// TwinCAT 3 PLC project MistralPLC
// ProgramVersion: 3.1.4023.0
// libraries:
//   Tc2_FTP, * (Beckhoff Automation GmbH)
//   Tc2_Standard, * (Beckhoff Automation GmbH)
//   Tc2_System, * (Beckhoff Automation GmbH)
//   Tc2_TcpIp, * (Beckhoff Automation GmbH)
//   Tc2_Utilities, * (Beckhoff Automation GmbH)
//   Tc3_EventLogger, * (Beckhoff Automation GmbH)
//   Tc3_Module, * (Beckhoff Automation GmbH)
//   Util, * (System)
// project tree:
//   Data types/ E_ClientSteps.TcDUT, E_DataExchaSteps.TcDUT
//   DUTs/ ST_LoadData.TcDUT
//   GVLs/Conveyor_1/ GVL_bButt_1.TcGVL, GVL_bDriveReady_1.TcGVL, GVL_bDrive_1.TcGVL, GVL_bLongMove_1.TcGVL, GVL_bMove_1.TcGVL, GVL_bPerm_1.TcGVL, GVL_bSens_1.TcGVL, GVL_BusyFree_1.TcGVL
//   GVLs/Conveyor_2/ GVL_bButt_2.TcGVL, GVL_bDriveReady_2.TcGVL, GVL_bDriveSpeed_2.TcGVL, GVL_bDrive_2.TcGVL, GVL_bLongMove_2.TcGVL, GVL_bMove_2.TcGVL, GVL_bPerm_2.TcGVL, GVL_bSens_2.TcGVL, GVL_BusyFree_2.TcGVL
//   GVLs/Conveyor_3/ GVL_bButt_3.TcGVL, GVL_bDriveReady_3.TcGVL, GVL_bDriveSpeed_3.TcGVL, GVL_bDrive_3.TcGVL, GVL_bLongMove_3.TcGVL, GVL_bMove_3.TcGVL, GVL_bPerm_3.TcGVL, GVL_bSens_3.TcGVL, GVL_BusyFree_3.TcGVL
//   GVLs/Conveyor_4/ GVL_bButt_4.TcGVL, GVL_bDriveReady_4.TcGVL, GVL_bDriveSpeed_4.TcGVL, GVL_bDrive_4.TcGVL, GVL_bLongMove_4.TcGVL, GVL_bMove_4.TcGVL, GVL_bPerm_4.TcGVL, GVL_bSens_4.TcGVL, GVL_BusyFree_4.TcGVL
//   GVLs/ Global_Variables.TcGVL, GVL.TcGVL, GVL_Alarm.TcGVL, GVL_Lights.TcGVL, GVL_LoadData_1.TcGVL
//   / PlcTask.TcTTO
//   POUs/Alarms/ AlarmEventGeneral.TcPOU, AlarmEvent_conv1.TcPOU, AlarmEvent_conv2.TcPOU, AlarmEvent_conv3.TcPOU, AlarmEvent_conv4.TcPOU, Alarm_conv_1.TcPOU, Alarm_conv_2.TcPOU, Alarm_conv_3.TcPOU, Alarm_conv_4.TcPOU, Alarm_conv_General.TcPOU, FB_AlarmEvent.TcPOU
//   POUs/ ConvLine1.TcPOU, ConvLine2.TcPOU, ConvLine3.TcPOU, ConvLine4.TcPOU, MAIN.TcPOU, TCP_IP.TcPOU
//   POUs/Ethernet/ FB_Server.TcPOU, FB_ServerApplication.TcPOU, FB_ServerConnection.TcPOU
//   POUs/Ethernet/Helper POUs/ FB_FrameFifo.TcPOU, FB_LogFifo.TcPOU
//   POUs/ExchangeWMS/ Exchange_WMS.TcPOU, FB_CreateMessage.TcPOU, FB_LoadDataToWMS.TcPOU, FB_Tail.TcPOU, FB_TransBuffer.TcPOU, FB_Upload_ToServer.TcPOU
//   POUs/FB/FBauxiliary/ FB_Busy1.TcPOU, FB_Busy2.TcPOU, FB_ButtonToggle.TcPOU
//   POUs/FB/FBconv/ FB_ConvPlace.TcPOU, FB_ConvPlaceDouble.TcPOU
//   POUs/FB/ FB_Direction.TcPOU, FB_Puls.TcPOU, Puls.TcPOU
//   POUs/ProcessingLoadData/ FB_LoadScan.TcPOU, FB_LoadWeight.TcPOU
// real-time tasks:
//   TASK PlcTask: cycle T#10ms, priority 20, ADS port 350
// I/O:
//   DEVICE Device 2 (Profinet Controller CCAT (RT)), AmsNetId 5.79.109.88.2.1
//     scale1 [BIZERBA BIZERBA Industrial weighing terminal WM4 920008000]
//       modules: Term 1 (DAP Module), Term 2 (Output 1 word), Term 3 (Output 1 byte), Term 4 (Output 1 byte), Term 5 (Output 1 byte), Term 6 (Output 1 byte), Term 7 (Output 1 byte), Term 8 (Output 1 byte), Term 9 (Output 1 byte), Term 10 (Output 1 byte), Term 11 (Output 1 byte), Term 12 (Output 1 byte), Term 13 (Output 1 byte), Term 14 (Output 1 byte), Term 15 (Output 1 byte), Term 16 (Output 1 byte), Term 17 (Input 1 word), Term 18 (Input 2 word), Term 19 (Input 1 byte), Term 20 (Input 1 byte), Term 21 (Input 1 byte), Term 22 (Input 1 byte), Term 23 (Input 1 byte), Term 24 (Input 1 byte), Term 25 (Input 1 byte), Term 26 (Input 1 byte), Term 27 (Input 1 byte), Term 28 (Input 1 byte)
//     scale2 [BIZERBA BIZERBA Industrial weighing terminal WM4 920008000]
//       modules: Term 31 (DAP Module), Term 86 (Output 1 word), Term 87 (Output 1 byte), Term 88 (Output 1 byte), Term 89 (Output 1 byte), Term 90 (Output 1 byte), Term 91 (Output 1 byte), Term 92 (Output 1 byte), Term 93 (Output 1 byte), Term 94 (Output 1 byte), Term 95 (Output 1 byte), Term 96 (Output 1 byte), Term 97 (Output 1 byte), Term 98 (Output 1 byte), Term 99 (Output 1 byte), Term 100 (Output 1 byte), Term 101 (Input 1 word), Term 102 (Input 2 word), Term 103 (Input 1 byte), Term 104 (Input 1 byte), Term 105 (Input 1 byte), Term 106 (Input 1 byte), Term 107 (Input 1 byte), Term 108 (Input 1 byte), Term 109 (Input 1 byte), Term 110 (Input 1 byte), Term 111 (Input 1 byte), Term 112 (Input 1 byte)
//     scale3 [BIZERBA BIZERBA Industrial weighing terminal WM4 920008000]
//       modules: Term 29 (DAP Module), Term 32 (Output 1 word), Term 33 (Output 1 byte), Term 34 (Output 1 byte), Term 35 (Output 1 byte), Term 36 (Output 1 byte), Term 37 (Output 1 byte), Term 38 (Output 1 byte), Term 39 (Output 1 byte), Term 40 (Output 1 byte), Term 41 (Output 1 byte), Term 42 (Output 1 byte), Term 43 (Output 1 byte), Term 44 (Output 1 byte), Term 45 (Output 1 byte), Term 46 (Output 1 byte), Term 47 (Input 1 word), Term 48 (Input 2 word), Term 49 (Input 1 byte), Term 50 (Input 1 byte), Term 51 (Input 1 byte), Term 52 (Input 1 byte), Term 53 (Input 1 byte), Term 54 (Input 1 byte), Term 55 (Input 1 byte), Term 56 (Input 1 byte), Term 57 (Input 1 byte), Term 58 (Input 1 byte)
//     scale4 [BIZERBA BIZERBA Industrial weighing terminal WM4 920008000]
//       modules: Term 30 (DAP Module), Term 59 (Output 1 word), Term 60 (Output 1 byte), Term 61 (Output 1 byte), Term 62 (Output 1 byte), Term 63 (Output 1 byte), Term 64 (Output 1 byte), Term 65 (Output 1 byte), Term 66 (Output 1 byte), Term 67 (Output 1 byte), Term 68 (Output 1 byte), Term 69 (Output 1 byte), Term 70 (Output 1 byte), Term 71 (Output 1 byte), Term 72 (Output 1 byte), Term 73 (Output 1 byte), Term 74 (Input 1 word), Term 75 (Input 2 word), Term 76 (Input 1 byte), Term 77 (Input 1 byte), Term 78 (Input 1 byte), Term 79 (Input 1 byte), Term 80 (Input 1 byte), Term 81 (Input 1 byte), Term 82 (Input 1 byte), Term 83 (Input 1 byte), Term 84 (Input 1 byte), Term 85 (Input 1 byte)
//   DEVICE Device 1 (EtherCAT), AmsNetId 5.79.109.88.3.1
//     Term 1 (EK1200) [EK1200-5000 EtherCAT Power supply (2A E-Bus)]
//       Term 2 (EL1008) [EL1008 8Ch. Dig. Input 24V, 3ms]
//       Term 3 (EL1008) [EL1008 8Ch. Dig. Input 24V, 3ms]
//       Term 4 (EL1008) [EL1008 8Ch. Dig. Input 24V, 3ms]
//       Term 5 (EL1008) [EL1008 8Ch. Dig. Input 24V, 3ms]
//       Term 6 (EL1008) [EL1008 8Ch. Dig. Input 24V, 3ms]
//       Term 7 (EL2008) [EL2008 8Ch. Dig. Output 24V, 0.5A]
//       Term 8 (EL2008) [EL2008 8Ch. Dig. Output 24V, 0.5A]
//       Term 9 (EL2008) [EL2008 8Ch. Dig. Output 24V, 0.5A]
//       Term 10 (EL2008) [EL2008 8Ch. Dig. Output 24V, 0.5A]
//       Term 11 (EK1122) [EK1122 2 port EtherCAT junction]
//         Term 12 (EK1100) [EK1100 EtherCAT Coupler (2A E-Bus)]
//           Term 15 (EL1008) [EL1008 8Ch. Dig. Input 24V, 3ms]
//           Term 16 (EL1008) [EL1008 8Ch. Dig. Input 24V, 3ms]
//           Term 17 (EL1008) [EL1008 8Ch. Dig. Input 24V, 3ms]
//           Term 18 (EL1008) [EL1008 8Ch. Dig. Input 24V, 3ms]
//           Term 19 (EL1008) [EL1008 8Ch. Dig. Input 24V, 3ms]
//           Term 20 (EL2008) [EL2008 8Ch. Dig. Output 24V, 0.5A]
//           Term 21 (EL2008) [EL2008 8Ch. Dig. Output 24V, 0.5A]
//           Term 22 (EL2008) [EL2008 8Ch. Dig. Output 24V, 0.5A]
//           Term 23 (EL2008) [EL2008 8Ch. Dig. Output 24V, 0.5A]
//           Term 24 (EK1322) [EK1322 2-port EtherCAT P junction with feed-in]
//             Box 1 (EPP2339-0021) X3 [EPP2339-0021 16 Ch. Dig. Input/Output 24V, 0,5A, M8]
//             Box 2 (EPP1004-0061) X3 [EPP1004-0061 4 Ch. Dig. Input 24V, 3ms, M8]
//             Box 3 (EPP2339-0021) X3 [EPP2339-0021 16 Ch. Dig. Input/Output 24V, 0,5A, M8]
//             Box 4 (EPP2339-0021) X4 [EPP2339-0021 16 Ch. Dig. Input/Output 24V, 0,5A, M8]
//             Box 5 (EPP1004-0061) X4 [EPP1004-0061 4 Ch. Dig. Input 24V, 3ms, M8]
//             Box 6 (EPP2339-0021) X4 [EPP2339-0021 16 Ch. Dig. Input/Output 24V, 0,5A, M8]
//       Term 13 (EK1322) [EK1322 2-port EtherCAT P junction with feed-in]
//         Box 1 (EPP2339-0021) X1 [EPP2339-0021 16 Ch. Dig. Input/Output 24V, 0,5A, M8]
//         Box 2 (EPP1004-0061) X1 [EPP1004-0061 4 Ch. Dig. Input 24V, 3ms, M8]
//         Box 3 (EPP2339-0021) X1 [EPP2339-0021 16 Ch. Dig. Input/Output 24V, 0,5A, M8]
//         Box 4 (EPP2339-0021) X2 [EPP2339-0021 16 Ch. Dig. Input/Output 24V, 0,5A, M8]
//         Box 5 (EPP1004-0061) X2 [EPP1004-0061 4 Ch. Dig. Input 24V, 3ms, M8]
//         Box 6 (EPP2339-0021) X2 [EPP2339-0021 16 Ch. Dig. Input/Output 24V, 0,5A, M8]
// variable links:
//   MistralPLC/MistralPLC Instance <-> Device 1 (EtherCAT)/Term 1 (EK1200)/Term 11 (EK1122)/Term 12 (EK1100)/Term 15 (EL1008)
//     PlcTask Inputs/GVL.b_3AS1 <-> Channel 3/Input
//     PlcTask Inputs/GVL.b_4AS1 <-> Channel 4/Input
//     PlcTask Inputs/GVL.b_K2_ <-> Channel 2/Input
//     PlcTask Inputs/GVL.b_SF3_ <-> Channel 1/Input
//   MistralPLC/MistralPLC Instance <-> Device 1 (EtherCAT)/Term 1 (EK1200)/Term 11 (EK1122)/Term 12 (EK1100)/Term 16 (EL1008)
//     PlcTask Inputs/GVL.b_3KM1_1 <-> Channel 2/Input
//     PlcTask Inputs/GVL.b_3KM1_2 <-> Channel 3/Input
//     PlcTask Inputs/GVL.b_4KM1_1 <-> Channel 5/Input
//     PlcTask Inputs/GVL.b_4KM1_2 <-> Channel 6/Input
//     PlcTask Inputs/GVL.b_3QF1 <-> Channel 1/Input
//     PlcTask Inputs/GVL.b_4QF1 <-> Channel 4/Input
//   MistralPLC/MistralPLC Instance <-> Device 1 (EtherCAT)/Term 1 (EK1200)/Term 11 (EK1122)/Term 12 (EK1100)/Term 17 (EL1008)
//     PlcTask Inputs/GVL.b_3KM{2..7} <-> Channel {3..8}/Input  (6 links)
//     PlcTask Inputs/GVL.b_3QF2_3QF7 <-> Channel 1/Input
//     PlcTask Inputs/GVL.b_3QF8 <-> Channel 2/Input
//   MistralPLC/MistralPLC Instance <-> Device 1 (EtherCAT)/Term 1 (EK1200)/Term 11 (EK1122)/Term 12 (EK1100)/Term 18 (EL1008)
//     PlcTask Inputs/GVL.b_4KM{2..7} <-> Channel {3..8}/Input  (6 links)
//     PlcTask Inputs/GVL.b_4QF2_4QF7 <-> Channel 1/Input
//     PlcTask Inputs/GVL.b_4QF8 <-> Channel 2/Input
//   MistralPLC/MistralPLC Instance <-> Device 1 (EtherCAT)/Term 1 (EK1200)/Term 11 (EK1122)/Term 12 (EK1100)/Term 20 (EL2008)
//     PlcTask Outputs/GVL.b3K{2..5} <-> Channel {5..8}/Output  (4 links)
//     PlcTask Outputs/GVL.b_3K1_1 <-> Channel 1/Output
//     PlcTask Outputs/GVL.b_3K1_2 <-> Channel 2/Output
//     PlcTask Outputs/GVL.b_4K1_1 <-> Channel 3/Output
//     PlcTask Outputs/GVL.b_4K1_2 <-> Channel 4/Output
//   MistralPLC/MistralPLC Instance <-> Device 1 (EtherCAT)/Term 1 (EK1200)/Term 11 (EK1122)/Term 12 (EK1100)/Term 21 (EL2008)
//     PlcTask Outputs/GVL.b3K6 <-> Channel 1/Output
//     PlcTask Outputs/GVL.b3K7 <-> Channel 2/Output
//     PlcTask Outputs/GVL.b4K2 <-> Channel 3/Output
//     PlcTask Outputs/GVL.b4K3 <-> Channel 4/Output
//     PlcTask Outputs/GVL.b4K4 <-> Channel 5/Output
//     PlcTask Outputs/GVL.b4K5 <-> Channel 6/Output
//     PlcTask Outputs/GVL.b4K6 <-> Channel 7/Output
//     PlcTask Outputs/GVL.b4K7 <-> Channel 8/Output
//   MistralPLC/MistralPLC Instance <-> Device 1 (EtherCAT)/Term 1 (EK1200)/Term 11 (EK1122)/Term 12 (EK1100)/Term 22 (EL2008)
//     PlcTask Outputs/GVL.b2Sh_SB0 <-> Channel 5/Output
//     PlcTask Outputs/GVL.b2Sh_SB1 <-> Channel 6/Output
//     PlcTask Outputs/GVL.b3S1_SB0 <-> Channel 1/Output
//     PlcTask Outputs/GVL.b3S6_SB0 <-> Channel 2/Output
//     PlcTask Outputs/GVL.b4S1_SB0 <-> Channel 3/Output
//     PlcTask Outputs/GVL.b4S6_SB0 <-> Channel 4/Output
//   MistralPLC/MistralPLC Instance <-> Device 1 (EtherCAT)/Term 1 (EK1200)/Term 11 (EK1122)/Term 12 (EK1100)/Term 24 (EK1322)/Box 1 (EPP2339-0021) X3
//     PlcTask Inputs/GVL.b3_S6_SB0 <-> Channel 11/Input
//     PlcTask Inputs/GVL_bSens_3.bSens3s04D1 <-> Channel 1/Input
//     PlcTask Inputs/GVL_bSens_3.bSens3s04D2 <-> Channel 2/Input
//     PlcTask Inputs/GVL_bSens_3.bSens3s04D3 <-> Channel 3/Input
//     PlcTask Inputs/GVL_bSens_3.bSens3s05D1 <-> Channel 4/Input
//     PlcTask Inputs/GVL_bSens_3.bSens3s05D2 <-> Channel 5/Input
//     PlcTask Inputs/GVL_bSens_3.bSens3s06D1 <-> Channel 6/Input
//     PlcTask Inputs/GVL_bSens_3.bSens3s06D2 <-> Channel 7/Input
//     PlcTask Outputs/GVL.b_3S4_2A2 <-> Channel 25/Output
//     PlcTask Outputs/GVL.b_3S5_2A1 <-> Channel 26/Output
//     PlcTask Outputs/GVL_Lights.bBlue_3S1HL1 <-> Channel 32/Output
//     PlcTask Outputs/GVL_Lights.bGreen_3S1HL1 <-> Channel 30/Output
//     PlcTask Outputs/GVL_Lights.bRed_3S1HL1 <-> Channel 29/Output
//     PlcTask Outputs/GVL_Lights.bSound_3S1HL1 <-> Channel 28/Output
//     PlcTask Outputs/GVL_Lights.bYellow_3S1HL1 <-> Channel 31/Output
//   MistralPLC/MistralPLC Instance <-> Device 1 (EtherCAT)/Term 1 (EK1200)/Term 11 (EK1122)/Term 12 (EK1100)/Term 24 (EK1322)/Box 2 (EPP1004-0061) X3
//     PlcTask Inputs/GVL_bSens_3.bSens3s02D1 <-> Channel 1/Input
//     PlcTask Inputs/GVL_bSens_3.bSens3s02D2 <-> Channel 2/Input
//     PlcTask Inputs/GVL_bSens_3.bSens3s03D1 <-> Channel 3/Input
//     PlcTask Inputs/GVL_bSens_3.bSens3s03D2 <-> Channel 4/Input
//   MistralPLC/MistralPLC Instance <-> Device 1 (EtherCAT)/Term 1 (EK1200)/Term 11 (EK1122)/Term 12 (EK1100)/Term 24 (EK1322)/Box 3 (EPP2339-0021) X3
//     PlcTask Inputs/GVL.b3_S1_SB0 <-> Channel 9/Input
//     PlcTask Inputs/GVL_bSens_3.bSens3s01D1 <-> Channel 1/Input
//     PlcTask Inputs/GVL_bSens_3.bSens3s01D2 <-> Channel 2/Input
//     PlcTask Inputs/GVL_bSens_3.bSens3s01D3 <-> Channel 3/Input
//     PlcTask Outputs/GVL_Lights.bBlue_3S1_HL1 <-> Channel 24/Output
//     PlcTask Outputs/GVL_Lights.bGreen_3S1_HL1 <-> Channel 22/Output
//     PlcTask Outputs/GVL_Lights.bRed_3S1_HL1 <-> Channel 21/Output
//     PlcTask Outputs/GVL_Lights.bSound_3S1_HL1 <-> Channel 20/Output
//     PlcTask Outputs/GVL_Lights.bYellow_3S1_HL1 <-> Channel 23/Output
//   MistralPLC/MistralPLC Instance <-> Device 1 (EtherCAT)/Term 1 (EK1200)/Term 11 (EK1122)/Term 12 (EK1100)/Term 24 (EK1322)/Box 4 (EPP2339-0021) X4
//     PlcTask Inputs/GVL.b4_S6_SB0 <-> Channel 11/Input
//     PlcTask Inputs/GVL_bSens_4.bSens4s04D1 <-> Channel 1/Input
//     PlcTask Inputs/GVL_bSens_4.bSens4s04D2 <-> Channel 2/Input
//     PlcTask Inputs/GVL_bSens_4.bSens4s04D3 <-> Channel 3/Input
//     PlcTask Inputs/GVL_bSens_4.bSens4s05D1 <-> Channel 4/Input
//     PlcTask Inputs/GVL_bSens_4.bSens4s05D2 <-> Channel 5/Input
//     PlcTask Inputs/GVL_bSens_4.bSens4s06D1 <-> Channel 6/Input
//     PlcTask Inputs/GVL_bSens_4.bSens4s06D2 <-> Channel 7/Input
//     PlcTask Outputs/GVL.b_4S4_2A2 <-> Channel 25/Output
//     PlcTask Outputs/GVL.b_4S5_2A1 <-> Channel 26/Output
//     PlcTask Outputs/GVL_Lights.bBlue_4S1HL1 <-> Channel 32/Output
//     PlcTask Outputs/GVL_Lights.bGreen_4S1HL1 <-> Channel 30/Output
//     PlcTask Outputs/GVL_Lights.bRed_4S1HL1 <-> Channel 24/Output
//     PlcTask Outputs/GVL_Lights.bSound_4S1HL1 <-> Channel 28/Output
//     PlcTask Outputs/GVL_Lights.bYellow_4S1HL1 <-> Channel 31/Output
//   MistralPLC/MistralPLC Instance <-> Device 1 (EtherCAT)/Term 1 (EK1200)/Term 11 (EK1122)/Term 12 (EK1100)/Term 24 (EK1322)/Box 5 (EPP1004-0061) X4
//     PlcTask Inputs/GVL_bSens_4.bSens4s02D1 <-> Channel 1/Input
//     PlcTask Inputs/GVL_bSens_4.bSens4s02D2 <-> Channel 2/Input
//     PlcTask Inputs/GVL_bSens_4.bSens4s03D1 <-> Channel 3/Input
//     PlcTask Inputs/GVL_bSens_4.bSens4s03D2 <-> Channel 4/Input
//   MistralPLC/MistralPLC Instance <-> Device 1 (EtherCAT)/Term 1 (EK1200)/Term 11 (EK1122)/Term 12 (EK1100)/Term 24 (EK1322)/Box 6 (EPP2339-0021) X4
//     PlcTask Inputs/GVL.b4_S1_SB0 <-> Channel 9/Input
//     PlcTask Inputs/GVL_bSens_4.bSens4s01D1 <-> Channel 1/Input
//     PlcTask Inputs/GVL_bSens_4.bSens4s01D2 <-> Channel 2/Input
//     PlcTask Inputs/GVL_bSens_4.bSens4s01D3 <-> Channel 3/Input
//     PlcTask Outputs/GVL_Lights.bBlue_4S1_HL1 <-> Channel 24/Output
//     PlcTask Outputs/GVL_Lights.bGreen_4S1_HL1 <-> Channel 22/Output
//     PlcTask Outputs/GVL_Lights.bRed_4S1_HL1 <-> Channel 21/Output
//     PlcTask Outputs/GVL_Lights.bSound_4S1_HL1 <-> Channel 20/Output
//     PlcTask Outputs/GVL_Lights.bYellow_4S1_HL1 <-> Channel 23/Output
//   MistralPLC/MistralPLC Instance <-> Device 1 (EtherCAT)/Term 1 (EK1200)/Term 13 (EK1322)/Box 1 (EPP2339-0021) X1
//     PlcTask Inputs/GVL.b1_S6_SB0 <-> Channel 11/Input
//     PlcTask Inputs/GVL_bSens_1.bSens1s04D1 <-> Channel 1/Input
//     PlcTask Inputs/GVL_bSens_1.bSens1s04D2 <-> Channel 2/Input
//     PlcTask Inputs/GVL_bSens_1.bSens1s04D3 <-> Channel 3/Input
//     PlcTask Inputs/GVL_bSens_1.bSens1s05D1 <-> Channel 4/Input
//     PlcTask Inputs/GVL_bSens_1.bSens1s05D2 <-> Channel 5/Input
//     PlcTask Inputs/GVL_bSens_1.bSens1s06D1 <-> Channel 6/Input
//     PlcTask Inputs/GVL_bSens_1.bSens1s06D2 <-> Channel 7/Input
//     PlcTask Outputs/GVL.b_1S4_2A2 <-> Channel 25/Output
//     PlcTask Outputs/GVL.b_1S5_2A1 <-> Channel 26/Output
//     PlcTask Outputs/GVL_Lights.bBlue_1S1HL1 <-> Channel 32/Output
//     PlcTask Outputs/GVL_Lights.bGreen_1S1HL1 <-> Channel 30/Output
//     PlcTask Outputs/GVL_Lights.bRed_1S1HL1 <-> Channel 29/Output
//     PlcTask Outputs/GVL_Lights.bSound_1S1HL1 <-> Channel 28/Output
//     PlcTask Outputs/GVL_Lights.bYellow_1S1HL1 <-> Channel 31/Output
//   MistralPLC/MistralPLC Instance <-> Device 1 (EtherCAT)/Term 1 (EK1200)/Term 13 (EK1322)/Box 2 (EPP1004-0061) X1
//     PlcTask Inputs/GVL_bSens_1.bSens1s02D1 <-> Channel 1/Input
//     PlcTask Inputs/GVL_bSens_1.bSens1s02D2 <-> Channel 2/Input
//     PlcTask Inputs/GVL_bSens_1.bSens1s03D1 <-> Channel 3/Input
//     PlcTask Inputs/GVL_bSens_1.bSens1s03D2 <-> Channel 4/Input
//   MistralPLC/MistralPLC Instance <-> Device 1 (EtherCAT)/Term 1 (EK1200)/Term 13 (EK1322)/Box 3 (EPP2339-0021) X1
//     PlcTask Inputs/GVL.b1_S1_SB0 <-> Channel 9/Input
//     PlcTask Inputs/GVL_bSens_1.bSens1s01D1 <-> Channel 1/Input
//     PlcTask Inputs/GVL_bSens_1.bSens1s01D2 <-> Channel 2/Input
//     PlcTask Inputs/GVL_bSens_1.bSens1s01D3 <-> Channel 3/Input
//     PlcTask Outputs/GVL_Lights.bBlue_1S1_HL1 <-> Channel 24/Output
//     PlcTask Outputs/GVL_Lights.bGreen_1S1_HL1 <-> Channel 22/Output
//     PlcTask Outputs/GVL_Lights.bRed_1S1_HL1 <-> Channel 21/Output
//     PlcTask Outputs/GVL_Lights.bSound_1S1_HL1 <-> Channel 20/Output
//     PlcTask Outputs/GVL_Lights.bYellow_1S1_HL1 <-> Channel 23/Output
//   MistralPLC/MistralPLC Instance <-> Device 1 (EtherCAT)/Term 1 (EK1200)/Term 13 (EK1322)/Box 4 (EPP2339-0021) X2
//     PlcTask Inputs/GVL.b2_S6_SB0 <-> Channel 11/Input
//     PlcTask Inputs/GVL_bSens_2.bSens2s04D1 <-> Channel 1/Input
//     PlcTask Inputs/GVL_bSens_2.bSens2s04D2 <-> Channel 2/Input
//     PlcTask Inputs/GVL_bSens_2.bSens2s04D3 <-> Channel 3/Input
//     PlcTask Inputs/GVL_bSens_2.bSens2s05D1 <-> Channel 4/Input
//     PlcTask Inputs/GVL_bSens_2.bSens2s05D2 <-> Channel 5/Input
//     PlcTask Inputs/GVL_bSens_2.bSens2s06D1 <-> Channel 6/Input
//     PlcTask Inputs/GVL_bSens_2.bSens2s06D2 <-> Channel 7/Input
//     PlcTask Outputs/GVL.b_2S4_2A2 <-> Channel 25/Output
//     PlcTask Outputs/GVL.b_2S5_2A1 <-> Channel 26/Output
//     PlcTask Outputs/GVL_Lights.bBlue_2S1HL1 <-> Channel 32/Output
//     PlcTask Outputs/GVL_Lights.bGreen_2S1HL1 <-> Channel 30/Output
//     PlcTask Outputs/GVL_Lights.bRed_2S1HL1 <-> Channel 29/Output
//     PlcTask Outputs/GVL_Lights.bSound_2S1HL1 <-> Channel 28/Output
//     PlcTask Outputs/GVL_Lights.bYellow_2S1HL1 <-> Channel 31/Output
//   MistralPLC/MistralPLC Instance <-> Device 1 (EtherCAT)/Term 1 (EK1200)/Term 13 (EK1322)/Box 5 (EPP1004-0061) X2
//     PlcTask Inputs/GVL_bSens_2.bSens2s02D1 <-> Channel 1/Input
//     PlcTask Inputs/GVL_bSens_2.bSens2s02D2 <-> Channel 2/Input
//     PlcTask Inputs/GVL_bSens_2.bSens2s03D1 <-> Channel 3/Input
//     PlcTask Inputs/GVL_bSens_2.bSens2s03D2 <-> Channel 4/Input
//   MistralPLC/MistralPLC Instance <-> Device 1 (EtherCAT)/Term 1 (EK1200)/Term 13 (EK1322)/Box 6 (EPP2339-0021) X2
//     PlcTask Inputs/GVL.b2_S1_SB0 <-> Channel 9/Input
//     PlcTask Inputs/GVL_bSens_2.bSens2s01D1 <-> Channel 1/Input
//     PlcTask Inputs/GVL_bSens_2.bSens2s01D2 <-> Channel 2/Input
//     PlcTask Inputs/GVL_bSens_2.bSens2s01D3 <-> Channel 3/Input
//     PlcTask Outputs/GVL_Lights.bBlue_2S1_HL1 <-> Channel 24/Output
//     PlcTask Outputs/GVL_Lights.bGreen_2S1_HL1 <-> Channel 22/Output
//     PlcTask Outputs/GVL_Lights.bRed_2S1_HL1 <-> Channel 21/Output
//     PlcTask Outputs/GVL_Lights.bSound_2S1_HL1 <-> Channel 20/Output
//     PlcTask Outputs/GVL_Lights.bYellow_2S1_HL1 <-> Channel 23/Output
//   MistralPLC/MistralPLC Instance <-> Device 1 (EtherCAT)/Term 1 (EK1200)/Term 2 (EL1008)
//     PlcTask Inputs/GVL.b_1AS1 <-> Channel 5/Input
//     PlcTask Inputs/GVL.b_2AS1 <-> Channel 6/Input
//     PlcTask Inputs/GVL.b_1QF <-> Channel 1/Input
//     PlcTask Inputs/GVL.b_2QF <-> Channel 2/Input
//     PlcTask Inputs/GVL.b_GP3 <-> Channel 7/Input
//     PlcTask Inputs/GVL.b_K2 <-> Channel 4/Input
//     PlcTask Inputs/GVL.b_SF3 <-> Channel 3/Input
//   MistralPLC/MistralPLC Instance <-> Device 1 (EtherCAT)/Term 1 (EK1200)/Term 3 (EL1008)
//     PlcTask Inputs/GVL.b_1KM1_1 <-> Channel 2/Input
//     PlcTask Inputs/GVL.b_1KM1_2 <-> Channel 3/Input
//     PlcTask Inputs/GVL.b_2KM1_1 <-> Channel 5/Input
//     PlcTask Inputs/GVL.b_2KM1_2 <-> Channel 6/Input
//     PlcTask Inputs/GVL.b_1P_I <-> Channel 7/Input
//     PlcTask Inputs/GVL.b_1P_U <-> Channel 8/Input
//     PlcTask Inputs/GVL.b_1QF1 <-> Channel 1/Input
//     PlcTask Inputs/GVL.b_2QF1 <-> Channel 4/Input
//   MistralPLC/MistralPLC Instance <-> Device 1 (EtherCAT)/Term 1 (EK1200)/Term 4 (EL1008)
//     PlcTask Inputs/GVL.b_1KM{2..7} <-> Channel {3..8}/Input  (6 links)
//     PlcTask Inputs/GVL.b_1QF2_1QF7 <-> Channel 1/Input
//     PlcTask Inputs/GVL.b_1QF8 <-> Channel 2/Input
//   MistralPLC/MistralPLC Instance <-> Device 1 (EtherCAT)/Term 1 (EK1200)/Term 5 (EL1008)
//     PlcTask Inputs/GVL.b_2KM{2..7} <-> Channel {3..8}/Input  (6 links)
//     PlcTask Inputs/GVL.b_2QF2_2QF7 <-> Channel 1/Input
//     PlcTask Inputs/GVL.b_2QF8 <-> Channel 2/Input
//   MistralPLC/MistralPLC Instance <-> Device 1 (EtherCAT)/Term 1 (EK1200)/Term 7 (EL2008)
//     PlcTask Outputs/GVL.b1K{2..5} <-> Channel {5..8}/Output  (4 links)
//     PlcTask Outputs/GVL.b_1K1_1 <-> Channel 1/Output
//     PlcTask Outputs/GVL.b_1K1_2 <-> Channel 2/Output
//     PlcTask Outputs/GVL.b_2K1_1 <-> Channel 3/Output
//     PlcTask Outputs/GVL.b_2K1_2 <-> Channel 4/Output
//   MistralPLC/MistralPLC Instance <-> Device 1 (EtherCAT)/Term 1 (EK1200)/Term 8 (EL2008)
//     PlcTask Outputs/GVL.b1K6 <-> Channel 1/Output
//     PlcTask Outputs/GVL.b1K7 <-> Channel 2/Output
//     PlcTask Outputs/GVL.b2K2 <-> Channel 3/Output
//     PlcTask Outputs/GVL.b2K3 <-> Channel 4/Output
//     PlcTask Outputs/GVL.b2K4 <-> Channel 5/Output
//     PlcTask Outputs/GVL.b2K5 <-> Channel 6/Output
//     PlcTask Outputs/GVL.b2K6 <-> Channel 7/Output
//     PlcTask Outputs/GVL.b2K7 <-> Channel 8/Output
//   MistralPLC/MistralPLC Instance <-> Device 1 (EtherCAT)/Term 1 (EK1200)/Term 9 (EL2008)
//     PlcTask Outputs/GVL.b1S1_SB0 <-> Channel 1/Output
//     PlcTask Outputs/GVL.b1S6_SB0 <-> Channel 2/Output
//     PlcTask Outputs/GVL.b2S1_SB0 <-> Channel 3/Output
//     PlcTask Outputs/GVL.b2S6_SB0 <-> Channel 4/Output
//     PlcTask Outputs/GVL.b1Sh_SB0 <-> Channel 5/Output
//     PlcTask Outputs/GVL.b1Sh_SB1 <-> Channel 6/Output
//   MistralPLC/MistralPLC Instance <-> Device 2 (Profinet Controller CCAT (RT))/scale1
//     PlcTask Inputs/GVL.Massa_1 <-> API/Term 18 (Input 2 word)/Subterm 21 (Input 2 word)/Inputs/Input
//   MistralPLC/MistralPLC Instance <-> Device 2 (Profinet Controller CCAT (RT))/scale2
//     PlcTask Inputs/GVL.Massa_2 <-> API/Term 102 (Input 2 word)/Subterm 114 (Input 2 word)/Inputs/Input
//   MistralPLC/MistralPLC Instance <-> Device 2 (Profinet Controller CCAT (RT))/scale3
//     PlcTask Inputs/GVL.Massa_3 <-> API/Term 48 (Input 2 word)/Subterm 60 (Input 2 word)/Inputs/Input
//   MistralPLC/MistralPLC Instance <-> Device 2 (Profinet Controller CCAT (RT))/scale4
//     PlcTask Inputs/GVL.Massa_4 <-> API/Term 75 (Input 2 word)/Subterm 87 (Input 2 word)/Inputs/Input

CONFIGURATION MistralPLC
    RESOURCE PLC ON TwinCAT3
        TASK PlcTask(INTERVAL := T#10ms, PRIORITY := 20);
        PROGRAM MAIN WITH PlcTask : MAIN;
    END_RESOURCE
END_CONFIGURATION

// ---- Data types/E_ClientSteps.TcDUT
TYPE E_ClientSteps :
(
	CLIENT_STATE_IDLE,
	CLIENT_STATE_CONNECT_START,
	CLIENT_STATE_CONNECT_WAIT,
	CLIENT_STATE_DATAEXCHA_START,
	CLIENT_STATE_DATAEXCHA_WAIT,
	CLIENT_STATE_CLOSE_START,
	CLIENT_STATE_CLOSE_WAIT,
	CLIENT_STATE_ERROR
);
END_TYPE

// ---- Data types/E_DataExchaSteps.TcDUT
TYPE E_DataExchaSteps :
(
	DATAEXCHA_STATE_IDLE,
	DATAEXCHA_STATE_SEND_START,
	DATAEXCHA_STATE_SEND_WAIT,
	DATAEXCHA_STATE_RECEIVE_START,
	DATAEXCHA_STATE_RECEIVE_WAIT,
	DATAEXCHA_STATE_ERROR
);
END_TYPE

// ---- DUTs/ST_LoadData.TcDUT
TYPE ST_LoadData :
STRUCT
	sID: STRING;
	sWeight: STRING;
END_STRUCT
END_TYPE

// ---- GVLs/Conveyor_1/GVL_bButt_1.TcGVL
VAR_GLOBAL
	bButtAuto1		:BOOL;
	bButtManu1		:BOOL;
	bButtStop1 		:BOOL;
	bButtReverse1 	:BOOL;
//-------------------------//
	bButt1s01		:BOOL;
	bButt1s01Rev	:BOOL;
	bButt1s02		:BOOL;
	bButt1s02Rev	:BOOL;
	bButt1s03		:BOOL;
	bButt1s03Rev	:BOOL;
	bButt1s04		:BOOL;
	bButt1s04Rev	:BOOL;								
	bButt1s05		:BOOL;									
	bButt1s05Rev	:BOOL;									
	bButt1s06		:BOOL;									
	bButt1s06Rev	:BOOL;
//-------------------------//
	bButt1s01_s02	:BOOL;
	bButt1s02_s03	:BOOL;
	bButt1s03_s04	:BOOL;
	bButt1s04_s05	:BOOL;
	bButt1s05_s06	:BOOL;

END_VAR

// ---- GVLs/Conveyor_1/GVL_bDriveReady_1.TcGVL
VAR_GLOBAL
// Готовность двигателей

bDriveReady1s01M1	AT%I* :BOOL;	// Конороль готовности конвейер 1 секция 1

bDriveReady1s02M1	AT%I* :BOOL;	// Конороль готовности конвейер 1 секция 2

bDriveReady1s03M1	AT%I* :BOOL;	// Конороль готовности конвейер 1 секция 3

bDriveReady1s04M1	AT%I* :BOOL;	// Конороль готовности конвейер 1 секция 4

bDriveReady1s05M1	AT%I* :BOOL;	// Конороль готовности конвейер 1 секция 5

bDriveReady1s06M1	AT%I* :BOOL;	// Конороль готовности конвейер 1 секция 6
END_VAR

// ---- GVLs/Conveyor_1/GVL_bDrive_1.TcGVL
VAR_GLOBAL

	bDrive1s01M1		  	 :BOOL;	
	bDrive1s01M1Rev	  		 :BOOL;

	bDrive1s02M1		  	 :BOOL;	
	bDrive1s02M1Rev	  		 :BOOL;

	bDrive1s03M1		  	 :BOOL;	
	bDrive1s03M1Rev	  		 :BOOL;

	bDrive1s04M1		  	 :BOOL;	
	bDrive1s04M1Rev	  		 :BOOL;

	bDrive1s05M1		  	 :BOOL;	
	bDrive1s05M1Rev	  		 :BOOL;

	bDrive1s06M1		  	 :BOOL;	
	bDrive1s06M1Rev	  		 :BOOL;
END_VAR

// ---- GVLs/Conveyor_1/GVL_bLongMove_1.TcGVL
VAR_GLOBAL
// Долгие перемещения
// Прямое движение	
bLongMove1s01_s02_1		:BOOL;
bLongMove1s02_1_s02_2   :BOOL;
bLongMove1s02_2_s03_1   :BOOL;
bLongMove1s02_s03       :BOOL;
bLongMove1s03_1_s03_2   :BOOL;
bLongMove1s03_2_s04_1   :BOOL;
bLongMove1s03_s04       :BOOL;
bLongMove1s04_1_s04_2   :BOOL;
bLongMove1s04_2_s05     :BOOL;
bLongMove1s05_1s06		:BOOL;

bLongMove_1s01_s02_1	 :BOOL;
bLongMove_1s02_1_s02_2   :BOOL;
bLongMove_1s02_2_s03_1   :BOOL;
bLongMove_1s02_s03       :BOOL;
bLongMove_1s03_1_s03_2   :BOOL;
bLongMove_1s03_2_s04_1   :BOOL;
bLongMove_1s03_s04       :BOOL;
bLongMove_1s04_1_s04_2   :BOOL;
bLongMove_1s04_2_s05     :BOOL;
bLongMove_1s05_1s06		:BOOL;  







END_VAR

// ---- GVLs/Conveyor_1/GVL_bMove_1.TcGVL
VAR_GLOBAL
// Прямое движение
bMove1s01_s02_1		:BOOL;
bMove1s02_1_s02_2	:BOOL;

bMove1s02_2_s03_1	:BOOL;
bMove1s02_s03		:BOOL;
bMove1s03_1_s03_2	:BOOL;

bMove1s03_2_s04_1	:BOOL;
bMove1s03_s04		:BOOL;
bMove1s04_1_s04_2	:BOOL;

bMove1s04_2_s05		:BOOL;
bMove1s05_s06		:BOOL;

END_VAR

// ---- GVLs/Conveyor_1/GVL_bPerm_1.TcGVL
VAR_GLOBAL
// Разрешение на движение
// Прямое движение
bPerm1s01_1s02	:BOOL;
bPerm1s02_1s03	:BOOL;
bPerm1s03_1s04	:BOOL;
bPerm1s04_1s05	:BOOL;
bPerm1s05_1s06	:BOOL;
// Обратное движение
bPerm1s06_1s05	:BOOL;
bPerm1s05_1s04	:BOOL;
bPerm1s04_1s03	:BOOL;
bPerm1s03_1s02	:BOOL;
bPerm1s02_1s01	:BOOL;
END_VAR

// ---- GVLs/Conveyor_1/GVL_bSens_1.TcGVL
VAR_GLOBAL
// --------------------------------------Список датчиков--------------------------------------------//
//---------------------------------------Первый конвейер--------------------------------------------//
{attribute 'TcLinkTo' := 'TIID^Device 1 (EtherCAT)^Term 1 (EK1200)^Term 13 (EK1322)^Box 3 (EPP2339-0021) X1^Channel 1^Input'}
bSens1s01D1 AT%I* :BOOL;	// Датчик в конце секции (в прямом направлении)
{attribute 'TcLinkTo' := 'TIID^Device 1 (EtherCAT)^Term 1 (EK1200)^Term 13 (EK1322)^Box 3 (EPP2339-0021) X1^Channel 2^Input'}
bSens1s01D2 AT%I* :BOOL;	// Датчик в конце секции (в обратном направлении)
{attribute 'TcLinkTo' := 'TIID^Device 1 (EtherCAT)^Term 1 (EK1200)^Term 13 (EK1322)^Box 3 (EPP2339-0021) X1^Channel 3^Input'}
bSens1s01D3 AT%I* :BOOL;	// Датчик контроля вил 
{attribute 'TcLinkTo' := 'TIID^Device 1 (EtherCAT)^Term 1 (EK1200)^Term 13 (EK1322)^Box 2 (EPP1004-0061) X1^Channel 1^Input'}
bSens1s02D1 AT%I* :BOOL;	// Датчик в конце секции (в прямом направлении)
{attribute 'TcLinkTo' := 'TIID^Device 1 (EtherCAT)^Term 1 (EK1200)^Term 13 (EK1322)^Box 2 (EPP1004-0061) X1^Channel 2^Input'}
bSens1s02D2 AT%I* :BOOL;	// Датчик в середине секции 
{attribute 'TcLinkTo' := 'TIID^Device 1 (EtherCAT)^Term 1 (EK1200)^Term 13 (EK1322)^Box 2 (EPP1004-0061) X1^Channel 3^Input'}
bSens1s03D1 AT%I* :BOOL;	// Датчик в конце секции (в прямом направлении)
{attribute 'TcLinkTo' := 'TIID^Device 1 (EtherCAT)^Term 1 (EK1200)^Term 13 (EK1322)^Box 2 (EPP1004-0061) X1^Channel 4^Input'}
bSens1s03D2 AT%I* :BOOL;	// Датчик в середине секции 
{attribute 'TcLinkTo' := 'TIID^Device 1 (EtherCAT)^Term 1 (EK1200)^Term 13 (EK1322)^Box 1 (EPP2339-0021) X1^Channel 1^Input'}
bSens1s04D1 AT%I* :BOOL;	// Датчик в конце секции (в прямом направлении)
{attribute 'TcLinkTo' := 'TIID^Device 1 (EtherCAT)^Term 1 (EK1200)^Term 13 (EK1322)^Box 1 (EPP2339-0021) X1^Channel 2^Input'}
bSens1s04D2 AT%I* :BOOL;	// Датчик в середине секции 
{attribute 'TcLinkTo' := 'TIID^Device 1 (EtherCAT)^Term 1 (EK1200)^Term 13 (EK1322)^Box 1 (EPP2339-0021) X1^Channel 3^Input'}
bSens1s04D3 AT%I* :BOOL;	// Датчик сканирования RFID
{attribute 'TcLinkTo' := 'TIID^Device 1 (EtherCAT)^Term 1 (EK1200)^Term 13 (EK1322)^Box 1 (EPP2339-0021) X1^Channel 4^Input'}
bSens1s05D1 AT%I* :BOOL;	// Датчик в конце секции (в прямом направлении)
{attribute 'TcLinkTo' := 'TIID^Device 1 (EtherCAT)^Term 1 (EK1200)^Term 13 (EK1322)^Box 1 (EPP2339-0021) X1^Channel 5^Input'}
bSens1s05D2 AT%I* :BOOL;	// Датчик управления двойным движением
{attribute 'TcLinkTo' := 'TIID^Device 1 (EtherCAT)^Term 1 (EK1200)^Term 13 (EK1322)^Box 1 (EPP2339-0021) X1^Channel 6^Input'}
bSens1s06D1 AT%I* :BOOL;	// Датчик в конце секции (в прямом направлении)
{attribute 'TcLinkTo' := 'TIID^Device 1 (EtherCAT)^Term 1 (EK1200)^Term 13 (EK1322)^Box 1 (EPP2339-0021) X1^Channel 7^Input'}
bSens1s06D2 AT%I* :BOOL;	// Датчик контроля вил

END_VAR

// ---- GVLs/Conveyor_1/GVL_BusyFree_1.TcGVL
VAR_GLOBAL
(*Текущее состояние платформы (Занято/Свободно)*)
(*Первый этаж*)
	bPlatformBusy1s01	 	:BOOL;
	bPlatformFree1s01 		:BOOL;
	bPlatformBusy1s02 		:BOOL;
	bPlatformFree1s02 		:BOOL;
	bPlatformBusy1s03 		:BOOL;
	bPlatformFree1s03 		:BOOL;
	bPlatformBusy1s04 		:BOOL;
	bPlatformFree1s04 		:BOOL;
	bPlatformBusy1s05		:BOOL;
	bPlatformFree1s05 		:BOOL;
	bPlatformBusy1s06		:BOOL;
	bPlatformFree1s06 		:BOOL;
END_VAR

// ---- GVLs/Conveyor_2/GVL_bButt_2.TcGVL
VAR_GLOBAL
	bButtAuto2		:BOOL;
	bButtManu2		:BOOL;
	bButtStop2 		:BOOL;
	bButtReverse2 	:BOOL;
//-------------------------//
	bButt2s01		:BOOL;
	bButt2s01Rev	:BOOL;
	bButt2s02		:BOOL;
	bButt2s02Rev	:BOOL;
	bButt2s03		:BOOL;
	bButt2s03Rev	:BOOL;
	bButt2s04		:BOOL;
	bButt2s04Rev	:BOOL;								
	bButt2s05		:BOOL;									
	bButt2s05Rev	:BOOL;									
	bButt2s06		:BOOL;									
	bButt2s06Rev	:BOOL;
//-------------------------//
	bButt2s01_s02	:BOOL;
	bButt2s02_s03	:BOOL;
	bButt2s03_s04	:BOOL;
	bButt2s04_s05	:BOOL;
	bButt2s05_s06	:BOOL;
END_VAR

// ---- GVLs/Conveyor_2/GVL_bDriveReady_2.TcGVL
VAR_GLOBAL
// Готовность двигателей

bDriveReady2s01M1	AT%I* :BOOL;	// Конороль готовности MoviMot конвейер 2 секция 1

bDriveReady2s02M1	AT%I* :BOOL;	// Конороль готовности MoviMot конвейер 2 секция 2

bDriveReady2s03M1	AT%I* :BOOL;	// Конороль готовности MoviMot конвейер 2 секция 3

bDriveReady2s04M1	AT%I* :BOOL;	// Конороль готовности MoviSwitch конвейер 2 секция 4

bDriveReady2s05M1	AT%I* :BOOL;	// Конороль готовности MoviSwitch конвейер 2 секция 5

bDriveReady2s06M1	AT%I* :BOOL;	// Конороль готовности MoviSwitch конвейер 2 секция 6
END_VAR

// ---- GVLs/Conveyor_2/GVL_bDriveSpeed_2.TcGVL
VAR_GLOBAL
// Включение второй скорости для секций

bDrive2s01Speed2			AT%Q* :BOOL;

bDrive2s02Speed2			AT%Q* :BOOL;

bDrive2s03Speed2			AT%Q* :BOOL;

bDrive2s04Speed2			AT%Q* :BOOL;

bDrive2s05Speed2			AT%Q* :BOOL;

bDrive2s06Speed2			AT%Q* :BOOL;
END_VAR

// ---- GVLs/Conveyor_2/GVL_bDrive_2.TcGVL
VAR_GLOBAL

	bDrive2s01M1		  	AT%Q* :BOOL;	
	bDrive2s01M1Rev	  		AT%Q* :BOOL;

	bDrive2s02M1		  	AT%Q* :BOOL;	
	bDrive2s02M1Rev	  		AT%Q* :BOOL;

	bDrive2s03M1		  	AT%Q* :BOOL;	
	bDrive2s03M1Rev	  		AT%Q* :BOOL;

	bDrive2s04M1		  	AT%Q* :BOOL;	
	bDrive2s04M1Rev	  		AT%Q* :BOOL;

	bDrive2s05M1		  	AT%Q* :BOOL;	
	bDrive2s05M1Rev	  		AT%Q* :BOOL;

	bDrive2s06M1		  	AT%Q* :BOOL;	
	bDrive2s06M1Rev	 	  	AT%Q* :BOOL;
END_VAR

// ---- GVLs/Conveyor_2/GVL_bLongMove_2.TcGVL
VAR_GLOBAL
// Долгие перемещения
// Прямое движение	
bLongMove2s01_s02_1		:BOOL;
bLongMove2s02_1_s02_2   :BOOL;
bLongMove2s02_2_s03_1   :BOOL;
bLongMove2s02_s03       :BOOL;
bLongMove2s03_1_s03_2   :BOOL;
bLongMove2s03_2_s04_1   :BOOL;
bLongMove2s03_s04       :BOOL;
bLongMove2s04_1_s04_2   :BOOL;
bLongMove2s04_2_s05     :BOOL;
bLongMove2s05_1s06		:BOOL;

bLongMove_2s01_s02_1	 :BOOL;
bLongMove_2s02_1_s02_2   :BOOL;
bLongMove_2s02_2_s03_1   :BOOL;
bLongMove_2s02_s03       :BOOL;
bLongMove_2s03_1_s03_2   :BOOL;
bLongMove_2s03_2_s04_1   :BOOL;
bLongMove_2s03_s04       :BOOL;
bLongMove_2s04_1_s04_2   :BOOL;
bLongMove_2s04_2_s05     :BOOL;
bLongMove_2s05_1s06		:BOOL;  
END_VAR

// ---- GVLs/Conveyor_2/GVL_bMove_2.TcGVL
VAR_GLOBAL
// Прямое движение
bMove2s01_s02_1		:BOOL;
bMove2s01_s02		:BOOL;
bMove2s02_1_s02_2	:BOOL;

bMove2s02_2_s03_1	:BOOL;
bMove2s02_s03		:BOOL;
bMove2s03_1_s03_2	:BOOL;

bMove2s03_2_s04_1	:BOOL;
bMove2s03_s04		:BOOL;
bMove2s04_1_s04_2	:BOOL;

bMove2s04_2_s05		:BOOL;
bMove2s05_s06		:BOOL;

END_VAR

// ---- GVLs/Conveyor_2/GVL_bPerm_2.TcGVL
VAR_GLOBAL
// Разрешение на движение
// Прямое движение
bPerm2s01_2s02	:BOOL;
bPerm2s02_2s03	:BOOL;
bPerm2s03_2s04	:BOOL;
bPerm2s04_2s05	:BOOL;
bPerm2s05_2s06	:BOOL;
// Обратное движение
bPerm2s06_2s05	:BOOL;
bPerm2s05_2s04	:BOOL;
bPerm2s04_2s03	:BOOL;
bPerm2s03_2s02	:BOOL;
bPerm2s02_2s01	:BOOL;
END_VAR

// ---- GVLs/Conveyor_2/GVL_bSens_2.TcGVL
VAR_GLOBAL
// --------------------------------------Список датчиков--------------------------------------------//
//---------------------------------------Второй конвейер--------------------------------------------//
{attribute 'TcLinkTo' := 'TIID^Device 1 (EtherCAT)^Term 1 (EK1200)^Term 13 (EK1322)^Box 6 (EPP2339-0021) X2^Channel 1^Input'}
bSens2s01D1 AT%I* :BOOL;	// Датчик в конце секции (в прямом направлении)
{attribute 'TcLinkTo' := 'TIID^Device 1 (EtherCAT)^Term 1 (EK1200)^Term 13 (EK1322)^Box 6 (EPP2339-0021) X2^Channel 2^Input'}
bSens2s01D2 AT%I* :BOOL;	// Датчик в конце секции (в обратном направлении
{attribute 'TcLinkTo' := 'TIID^Device 1 (EtherCAT)^Term 1 (EK1200)^Term 13 (EK1322)^Box 6 (EPP2339-0021) X2^Channel 3^Input'}
bSens2s01D3 AT%I* :BOOL;	// Датчик контроля вил)
{attribute 'TcLinkTo' := 'TIID^Device 1 (EtherCAT)^Term 1 (EK1200)^Term 13 (EK1322)^Box 5 (EPP1004-0061) X2^Channel 1^Input'}
bSens2s02D1 AT%I* :BOOL;	// Датчик в конце секции (в прямом направлении)
{attribute 'TcLinkTo' := 'TIID^Device 1 (EtherCAT)^Term 1 (EK1200)^Term 13 (EK1322)^Box 5 (EPP1004-0061) X2^Channel 2^Input'}
bSens2s02D2 AT%I* :BOOL;	// Датчик в середине секции 
{attribute 'TcLinkTo' := 'TIID^Device 1 (EtherCAT)^Term 1 (EK1200)^Term 13 (EK1322)^Box 5 (EPP1004-0061) X2^Channel 3^Input'}
bSens2s03D1 AT%I* :BOOL;	// Датчик в конце секции (в прямом направлении)
{attribute 'TcLinkTo' := 'TIID^Device 1 (EtherCAT)^Term 1 (EK1200)^Term 13 (EK1322)^Box 5 (EPP1004-0061) X2^Channel 4^Input'}
bSens2s03D2 AT%I* :BOOL;	// Датчик в середине секции 
{attribute 'TcLinkTo' := 'TIID^Device 1 (EtherCAT)^Term 1 (EK1200)^Term 13 (EK1322)^Box 4 (EPP2339-0021) X2^Channel 1^Input'}
bSens2s04D1 AT%I* :BOOL;	// Датчик в конце секции (в прямом направлении)
{attribute 'TcLinkTo' := 'TIID^Device 1 (EtherCAT)^Term 1 (EK1200)^Term 13 (EK1322)^Box 4 (EPP2339-0021) X2^Channel 2^Input'}
bSens2s04D2 AT%I* :BOOL;	// Датчик в середине секции 
{attribute 'TcLinkTo' := 'TIID^Device 1 (EtherCAT)^Term 1 (EK1200)^Term 13 (EK1322)^Box 4 (EPP2339-0021) X2^Channel 3^Input'}
bSens2s04D3 AT%I* :BOOL;	// Датчик сканирования RFID
{attribute 'TcLinkTo' := 'TIID^Device 1 (EtherCAT)^Term 1 (EK1200)^Term 13 (EK1322)^Box 4 (EPP2339-0021) X2^Channel 4^Input'}
bSens2s05D1 AT%I* :BOOL;	// Датчик в конце секции (в прямом направлении)
{attribute 'TcLinkTo' := 'TIID^Device 1 (EtherCAT)^Term 1 (EK1200)^Term 13 (EK1322)^Box 4 (EPP2339-0021) X2^Channel 5^Input'}
bSens2s05D2 AT%I* :BOOL;	// Датчик управления двойным движением
{attribute 'TcLinkTo' := 'TIID^Device 1 (EtherCAT)^Term 1 (EK1200)^Term 13 (EK1322)^Box 4 (EPP2339-0021) X2^Channel 6^Input'}
bSens2s06D1 AT%I* :BOOL;	// Датчик в конце секции (в прямом направлении)
{attribute 'TcLinkTo' := 'TIID^Device 1 (EtherCAT)^Term 1 (EK1200)^Term 13 (EK1322)^Box 4 (EPP2339-0021) X2^Channel 7^Input'}
bSens2s06D2 AT%I* :BOOL;	// Датчик контроля вил

END_VAR

// ---- GVLs/Conveyor_2/GVL_BusyFree_2.TcGVL
VAR_GLOBAL
(*Текущее состояние платформы (Занято/Свободно)*)
(*Первый этаж*)
	bPlatformBusy2s01	 	:BOOL;
	bPlatformFree2s01 		:BOOL;
	bPlatformBusy2s02 		:BOOL;
	bPlatformFree2s02 		:BOOL;
	bPlatformBusy2s03 		:BOOL;
	bPlatformFree2s03 		:BOOL;
	bPlatformBusy2s04 		:BOOL;
	bPlatformFree2s04 		:BOOL;
	bPlatformBusy2s05		:BOOL;
	bPlatformFree2s05 		:BOOL;
	bPlatformBusy2s06		:BOOL;
	bPlatformFree2s06 		:BOOL;
END_VAR

// ---- GVLs/Conveyor_3/GVL_bButt_3.TcGVL
VAR_GLOBAL
	bButtAuto3		:BOOL;
	bButtManu3		:BOOL;
	bButtStop3 		:BOOL;
	bButtReverse3 	:BOOL;
//-------------------------//
	bButt3s01		:BOOL;
	bButt3s01Rev	:BOOL;
	bButt3s02		:BOOL;
	bButt3s02Rev	:BOOL;
	bButt3s03		:BOOL;
	bButt3s03Rev	:BOOL;
	bButt3s04		:BOOL;
	bButt3s04Rev	:BOOL;								
	bButt3s05		:BOOL;									
	bButt3s05Rev	:BOOL;									
	bButt3s06		:BOOL;									
	bButt3s06Rev	:BOOL;
//-------------------------//
	bButt3s01_s02	:BOOL;
	bButt3s02_s03	:BOOL;
	bButt3s03_s04	:BOOL;
	bButt3s04_s05	:BOOL;
	bButt3s05_s06	:BOOL;
END_VAR

// ---- GVLs/Conveyor_3/GVL_bDriveReady_3.TcGVL
VAR_GLOBAL
// Готовность двигателей

bDriveReady3s01M1	AT%I* :BOOL;	// Конороль готовности MoviMot конвейер 3 секция 1

bDriveReady3s02M1	AT%I* :BOOL;	// Конороль готовности MoviMot конвейер 3 секция 2

bDriveReady3s03M1	AT%I* :BOOL;	// Конороль готовности MoviMot конвейер 3 секция 3

bDriveReady3s04M1	AT%I* :BOOL;	// Конороль готовности MoviSwitch конвейер 3 секция 4

bDriveReady3s05M1	AT%I* :BOOL;	// Конороль готовности MoviSwitch конвейер 3 секция 5

bDriveReady3s06M1	AT%I* :BOOL;	// Конороль готовности MoviSwitch конвейер 3 секция 6
END_VAR

// ---- GVLs/Conveyor_3/GVL_bDriveSpeed_3.TcGVL
VAR_GLOBAL
// Включение второй скорости для секций

bDrive3s01Speed2			AT%Q* :BOOL;

bDrive3s02Speed2			AT%Q* :BOOL;

bDrive3s03Speed2			AT%Q* :BOOL;

bDrive3s04Speed2			AT%Q* :BOOL;

bDrive3s05Speed2			AT%Q* :BOOL;

bDrive3s06Speed2			AT%Q* :BOOL;
END_VAR

// ---- GVLs/Conveyor_3/GVL_bDrive_3.TcGVL
VAR_GLOBAL

	bDrive3s01M1		  	AT%Q* :BOOL;	
	bDrive3s01M1Rev	  		AT%Q* :BOOL;

	bDrive3s02M1		  	AT%Q* :BOOL;	
	bDrive3s02M1Rev	  		AT%Q* :BOOL;

	bDrive3s03M1		  	AT%Q* :BOOL;	
	bDrive3s03M1Rev	  		AT%Q* :BOOL;

	bDrive3s04M1		  	AT%Q* :BOOL;	
	bDrive3s04M1Rev	  		AT%Q* :BOOL;

	bDrive3s05M1		  	AT%Q* :BOOL;	
	bDrive3s05M1Rev	  		AT%Q* :BOOL;

	bDrive3s06M1		  	AT%Q* :BOOL;	
	bDrive3s06M1Rev	 	  	AT%Q* :BOOL;
END_VAR

// ---- GVLs/Conveyor_3/GVL_bLongMove_3.TcGVL
VAR_GLOBAL
// Долгие перемещения
// Прямое движение	
bLongMove3s01_s02_1		:BOOL;
bLongMove3s02_1_s02_2   :BOOL;
bLongMove3s02_2_s03_1   :BOOL;
bLongMove3s02_s03       :BOOL;
bLongMove3s03_1_s03_2   :BOOL;
bLongMove3s03_2_s04_1   :BOOL;
bLongMove3s03_s04       :BOOL;
bLongMove3s04_1_s04_2   :BOOL;
bLongMove3s04_2_s05     :BOOL;
bLongMove3s05_1s06		:BOOL;

bLongMove_3s01_s02_1	 :BOOL;
bLongMove_3s02_1_s02_2   :BOOL;
bLongMove_3s02_2_s03_1   :BOOL;
bLongMove_3s02_s03       :BOOL;
bLongMove_3s03_1_s03_2   :BOOL;
bLongMove_3s03_2_s04_1   :BOOL;
bLongMove_3s03_s04       :BOOL;
bLongMove_3s04_1_s04_2   :BOOL;
bLongMove_3s04_2_s05     :BOOL;
bLongMove_3s05_1s06		:BOOL;  
END_VAR

// ---- GVLs/Conveyor_3/GVL_bMove_3.TcGVL
VAR_GLOBAL
// Прямое движение
bMove3s01_s02_1		:BOOL;
bMove3s02_1_s02_2	:BOOL;

bMove3s02_2_s03_1	:BOOL;
bMove3s02_s03		:BOOL;
bMove3s03_1_s03_2	:BOOL;

bMove3s03_2_s04_1	:BOOL;
bMove3s03_s04		:BOOL;
bMove3s04_1_s04_2	:BOOL;

bMove3s04_2_s05		:BOOL;
bMove3s05_s06		:BOOL;
END_VAR

// ---- GVLs/Conveyor_3/GVL_bPerm_3.TcGVL
VAR_GLOBAL
// Разрешение на движение
// Прямое движение
bPerm3s01_3s02	:BOOL;
bPerm3s02_3s03	:BOOL;
bPerm3s03_3s04	:BOOL;
bPerm3s04_3s05	:BOOL;
bPerm3s05_3s06	:BOOL;
// Обратное движение
bPerm3s06_3s05	:BOOL;
bPerm3s05_3s04	:BOOL;
bPerm3s04_3s03	:BOOL;
bPerm3s03_3s02	:BOOL;
bPerm3s02_3s01	:BOOL;
END_VAR

// ---- GVLs/Conveyor_3/GVL_bSens_3.TcGVL
VAR_GLOBAL
// --------------------------------------Список датчиков--------------------------------------------//
//---------------------------------------Третий конвейер--------------------------------------------//
{attribute 'TcLinkTo' := 'TIID^Device 1 (EtherCAT)^Term 1 (EK1200)^Term 11 (EK1122)^Term 12 (EK1100)^Term 24 (EK1322)^Box 3 (EPP2339-0021) X3^Channel 1^Input'}
bSens3s01D1 AT%I* :BOOL;	// Датчик в конце секции (в прямом направлении)
{attribute 'TcLinkTo' := 'TIID^Device 1 (EtherCAT)^Term 1 (EK1200)^Term 11 (EK1122)^Term 12 (EK1100)^Term 24 (EK1322)^Box 3 (EPP2339-0021) X3^Channel 2^Input'}
bSens3s01D2 AT%I* :BOOL;	// Датчик в конце секции (в обратном направлении) 
{attribute 'TcLinkTo' := 'TIID^Device 1 (EtherCAT)^Term 1 (EK1200)^Term 11 (EK1122)^Term 12 (EK1100)^Term 24 (EK1322)^Box 3 (EPP2339-0021) X3^Channel 3^Input'}
bSens3s01D3 AT%I* :BOOL;	// Датчик контроля вил
{attribute 'TcLinkTo' := 'TIID^Device 1 (EtherCAT)^Term 1 (EK1200)^Term 11 (EK1122)^Term 12 (EK1100)^Term 24 (EK1322)^Box 2 (EPP1004-0061) X3^Channel 1^Input'}
bSens3s02D1 AT%I* :BOOL;	// Датчик в конце секции (в прямом направлении)
{attribute 'TcLinkTo' := 'TIID^Device 1 (EtherCAT)^Term 1 (EK1200)^Term 11 (EK1122)^Term 12 (EK1100)^Term 24 (EK1322)^Box 2 (EPP1004-0061) X3^Channel 2^Input'}
bSens3s02D2 AT%I* :BOOL;	// Датчик в середине секции 
{attribute 'TcLinkTo' := 'TIID^Device 1 (EtherCAT)^Term 1 (EK1200)^Term 11 (EK1122)^Term 12 (EK1100)^Term 24 (EK1322)^Box 2 (EPP1004-0061) X3^Channel 3^Input'}
bSens3s03D1 AT%I* :BOOL;	// Датчик в конце секции (в прямом направлении)
{attribute 'TcLinkTo' := 'TIID^Device 1 (EtherCAT)^Term 1 (EK1200)^Term 11 (EK1122)^Term 12 (EK1100)^Term 24 (EK1322)^Box 2 (EPP1004-0061) X3^Channel 4^Input'}
bSens3s03D2 AT%I* :BOOL;	// Датчик в середине секции 
{attribute 'TcLinkTo' := 'TIID^Device 1 (EtherCAT)^Term 1 (EK1200)^Term 11 (EK1122)^Term 12 (EK1100)^Term 24 (EK1322)^Box 1 (EPP2339-0021) X3^Channel 1^Input'}
bSens3s04D1 AT%I* :BOOL;	// Датчик в конце секции (в прямом направлении)
{attribute 'TcLinkTo' := 'TIID^Device 1 (EtherCAT)^Term 1 (EK1200)^Term 11 (EK1122)^Term 12 (EK1100)^Term 24 (EK1322)^Box 1 (EPP2339-0021) X3^Channel 2^Input'}
bSens3s04D2 AT%I* :BOOL;	// Датчик в середине секции 
{attribute 'TcLinkTo' := 'TIID^Device 1 (EtherCAT)^Term 1 (EK1200)^Term 11 (EK1122)^Term 12 (EK1100)^Term 24 (EK1322)^Box 1 (EPP2339-0021) X3^Channel 3^Input'}
bSens3s04D3 AT%I* :BOOL;	// Датчик сканирования RFID
{attribute 'TcLinkTo' := 'TIID^Device 1 (EtherCAT)^Term 1 (EK1200)^Term 11 (EK1122)^Term 12 (EK1100)^Term 24 (EK1322)^Box 1 (EPP2339-0021) X3^Channel 4^Input'}
bSens3s05D1 AT%I* :BOOL;	// Датчик в конце секции (в прямом направлении)
{attribute 'TcLinkTo' := 'TIID^Device 1 (EtherCAT)^Term 1 (EK1200)^Term 11 (EK1122)^Term 12 (EK1100)^Term 24 (EK1322)^Box 1 (EPP2339-0021) X3^Channel 5^Input'}
bSens3s05D2 AT%I* :BOOL;	// Датчик управления двойным движением
{attribute 'TcLinkTo' := 'TIID^Device 1 (EtherCAT)^Term 1 (EK1200)^Term 11 (EK1122)^Term 12 (EK1100)^Term 24 (EK1322)^Box 1 (EPP2339-0021) X3^Channel 6^Input'}
bSens3s06D1 AT%I* :BOOL;	// Датчик в конце секции (в прямом направлении)
{attribute 'TcLinkTo' := 'TIID^Device 1 (EtherCAT)^Term 1 (EK1200)^Term 11 (EK1122)^Term 12 (EK1100)^Term 24 (EK1322)^Box 1 (EPP2339-0021) X3^Channel 7^Input'}
bSens3s06D2 AT%I* :BOOL;	// Датчик контроля вил

END_VAR

// ---- GVLs/Conveyor_3/GVL_BusyFree_3.TcGVL
VAR_GLOBAL
(*Текущее состояние платформы (Занято/Свободно)*)
(*Первый этаж*)
	bPlatformBusy3s01	 	:BOOL;
	bPlatformFree3s01 		:BOOL;
	bPlatformBusy3s02 		:BOOL;
	bPlatformFree3s02 		:BOOL;
	bPlatformBusy3s03 		:BOOL;
	bPlatformFree3s03 		:BOOL;
	bPlatformBusy3s04 		:BOOL;
	bPlatformFree3s04 		:BOOL;
	bPlatformBusy3s05		:BOOL;
	bPlatformFree3s05 		:BOOL;
	bPlatformBusy3s06		:BOOL;
	bPlatformFree3s06 		:BOOL;
END_VAR

// ---- GVLs/Conveyor_4/GVL_bButt_4.TcGVL
VAR_GLOBAL
	bButtAuto4		:BOOL;
	bButtManu4		:BOOL;
	bButtStop4 		:BOOL;
	bButtReverse4 	:BOOL;
//--------------------------//
	bButt4s01		:BOOL;
	bButt4s01Rev	:BOOL;
	bButt4s02		:BOOL;
	bButt4s02Rev	:BOOL;
	bButt4s03		:BOOL;
	bButt4s03Rev	:BOOL;
	bButt4s04		:BOOL;
	bButt4s04Rev	:BOOL;								
	bButt4s05		:BOOL;									
	bButt4s05Rev	:BOOL;									
	bButt4s06		:BOOL;									
	bButt4s06Rev	:BOOL;
//--------------------------//
	bButt4s01_s02	:BOOL;
	bButt4s02_s03	:BOOL;
	bButt4s03_s04	:BOOL;
	bButt4s04_s05	:BOOL;
	bButt4s05_s06	:BOOL;
END_VAR

// ---- GVLs/Conveyor_4/GVL_bDriveReady_4.TcGVL
VAR_GLOBAL
// Готовность двигателей

bDriveReady4s01M1	AT%I* :BOOL;	// Конороль готовности MoviMot конвейер 4 секция 1

bDriveReady4s02M1	AT%I* :BOOL;	// Конороль готовности MoviMot конвейер 4 секция 2

bDriveReady4s03M1	AT%I* :BOOL;	// Конороль готовности MoviMot конвейер 4 секция 3

bDriveReady4s04M1	AT%I* :BOOL;	// Конороль готовности MoviSwitch конвейер 4 секция 4

bDriveReady4s05M1	AT%I* :BOOL;	// Конороль готовности MoviSwitch конвейер 4 секция 5

bDriveReady4s06M1	AT%I* :BOOL;	// Конороль готовности MoviSwitch конвейер 4 секция 6
END_VAR

// ---- GVLs/Conveyor_4/GVL_bDriveSpeed_4.TcGVL
VAR_GLOBAL
// Включение второй скорости для секций

bDrive4s01Speed2			AT%Q* :BOOL;

bDrive4s02Speed2			AT%Q* :BOOL;

bDrive4s03Speed2			AT%Q* :BOOL;

bDrive4s04Speed2			AT%Q* :BOOL;

bDrive4s05Speed2			AT%Q* :BOOL;

bDrive4s06Speed2			AT%Q* :BOOL;
END_VAR

// ---- GVLs/Conveyor_4/GVL_bDrive_4.TcGVL
VAR_GLOBAL

	bDrive4s01M1		  	AT%Q* :BOOL;	
	bDrive4s01M1Rev	  		AT%Q* :BOOL;

	bDrive4s02M1		  	AT%Q* :BOOL;	
	bDrive4s02M1Rev	  		AT%Q* :BOOL;

	bDrive4s03M1		  	AT%Q* :BOOL;	
	bDrive4s03M1Rev	  		AT%Q* :BOOL;

	bDrive4s04M1		  	AT%Q* :BOOL;	
	bDrive4s04M1Rev	  		AT%Q* :BOOL;

	bDrive4s05M1		  	AT%Q* :BOOL;	
	bDrive4s05M1Rev	  		AT%Q* :BOOL;

	bDrive4s06M1		  	AT%Q* :BOOL;	
	bDrive4s06M1Rev	 	  	AT%Q* :BOOL;
END_VAR

// ---- GVLs/Conveyor_4/GVL_bLongMove_4.TcGVL
VAR_GLOBAL
// Долгие перемещения
// Прямое движение	
bLongMove4s01_s02_1		:BOOL;
bLongMove4s02_1_s02_2   :BOOL;
bLongMove4s02_2_s03_1   :BOOL;
bLongMove4s02_s03       :BOOL;
bLongMove4s03_1_s03_2   :BOOL;
bLongMove4s03_2_s04_1   :BOOL;
bLongMove4s03_s04       :BOOL;
bLongMove4s04_1_s04_2   :BOOL;
bLongMove4s04_2_s05     :BOOL;
bLongMove4s05_1s06		:BOOL;

bLongMove_4s01_s02_1	 :BOOL;
bLongMove_4s02_1_s02_2   :BOOL;
bLongMove_4s02_2_s03_1   :BOOL;
bLongMove_4s02_s03       :BOOL;
bLongMove_4s03_1_s03_2   :BOOL;
bLongMove_4s03_2_s04_1   :BOOL;
bLongMove_4s03_s04       :BOOL;
bLongMove_4s04_1_s04_2   :BOOL;
bLongMove_4s04_2_s05     :BOOL;
bLongMove_4s05_1s06		:BOOL;  
END_VAR

// ---- GVLs/Conveyor_4/GVL_bMove_4.TcGVL
VAR_GLOBAL
// Прямое движение
bMove4s01_s02_1		:BOOL;
bMove4s02_1_s02_2	:BOOL;

bMove4s02_2_s03_1	:BOOL;
bMove4s02_s03		:BOOL;
bMove4s03_1_s03_2	:BOOL;

bMove4s03_2_s04_1	:BOOL;
bMove4s03_s04		:BOOL;
bMove4s04_1_s04_2	:BOOL;

bMove4s04_2_s05		:BOOL;
bMove4s05_s06		:BOOL;
END_VAR

// ---- GVLs/Conveyor_4/GVL_bPerm_4.TcGVL
VAR_GLOBAL
// Разрешение на движение
// Прямое движение
bPerm4s01_4s02	:BOOL;
bPerm4s02_4s03	:BOOL;
bPerm4s03_4s04	:BOOL;
bPerm4s04_4s05	:BOOL;
bPerm4s05_4s06	:BOOL;
// Обратное движение
bPerm4s06_4s05	:BOOL;
bPerm4s05_4s04	:BOOL;
bPerm4s04_4s03	:BOOL;
bPerm4s03_4s02	:BOOL;
bPerm4s02_4s01	:BOOL;
END_VAR

// ---- GVLs/Conveyor_4/GVL_bSens_4.TcGVL
VAR_GLOBAL
// --------------------------------------Список датчиков--------------------------------------------//
//---------------------------------------Четвертый конвейер-----------------------------------------//
{attribute 'TcLinkTo' := 'TIID^Device 1 (EtherCAT)^Term 1 (EK1200)^Term 11 (EK1122)^Term 12 (EK1100)^Term 24 (EK1322)^Box 6 (EPP2339-0021) X4^Channel 1^Input'}
bSens4s01D1 AT%I* :BOOL;	// Датчик в конце секции (в прямом направлении)
{attribute 'TcLinkTo' := 'TIID^Device 1 (EtherCAT)^Term 1 (EK1200)^Term 11 (EK1122)^Term 12 (EK1100)^Term 24 (EK1322)^Box 6 (EPP2339-0021) X4^Channel 2^Input'}
bSens4s01D2 AT%I* :BOOL;	// Датчик в конце секции (в обратном направлении)
{attribute 'TcLinkTo' := 'TIID^Device 1 (EtherCAT)^Term 1 (EK1200)^Term 11 (EK1122)^Term 12 (EK1100)^Term 24 (EK1322)^Box 6 (EPP2339-0021) X4^Channel 3^Input'}
bSens4s01D3 AT%I* :BOOL;	// Датчик контроля вил 
{attribute 'TcLinkTo' := 'TIID^Device 1 (EtherCAT)^Term 1 (EK1200)^Term 11 (EK1122)^Term 12 (EK1100)^Term 24 (EK1322)^Box 5 (EPP1004-0061) X4^Channel 1^Input'}
bSens4s02D1 AT%I* :BOOL;	// Датчик в конце секции (в прямом направлении)
{attribute 'TcLinkTo' := 'TIID^Device 1 (EtherCAT)^Term 1 (EK1200)^Term 11 (EK1122)^Term 12 (EK1100)^Term 24 (EK1322)^Box 5 (EPP1004-0061) X4^Channel 2^Input'}
bSens4s02D2 AT%I* :BOOL;	// Датчик в середине секции 
{attribute 'TcLinkTo' := 'TIID^Device 1 (EtherCAT)^Term 1 (EK1200)^Term 11 (EK1122)^Term 12 (EK1100)^Term 24 (EK1322)^Box 5 (EPP1004-0061) X4^Channel 3^Input'}
bSens4s03D1 AT%I* :BOOL;	// Датчик в конце секции (в прямом направлении)
{attribute 'TcLinkTo' := 'TIID^Device 1 (EtherCAT)^Term 1 (EK1200)^Term 11 (EK1122)^Term 12 (EK1100)^Term 24 (EK1322)^Box 5 (EPP1004-0061) X4^Channel 4^Input'}
bSens4s03D2 AT%I* :BOOL;	// Датчик в середине секции 
{attribute 'TcLinkTo' := 'TIID^Device 1 (EtherCAT)^Term 1 (EK1200)^Term 11 (EK1122)^Term 12 (EK1100)^Term 24 (EK1322)^Box 4 (EPP2339-0021) X4^Channel 1^Input'}
bSens4s04D1 AT%I* :BOOL;	// Датчик в конце секции (в прямом направлении)
{attribute 'TcLinkTo' := 'TIID^Device 1 (EtherCAT)^Term 1 (EK1200)^Term 11 (EK1122)^Term 12 (EK1100)^Term 24 (EK1322)^Box 4 (EPP2339-0021) X4^Channel 2^Input'}
bSens4s04D2 AT%I* :BOOL;	// Датчик в середине секции 
{attribute 'TcLinkTo' := 'TIID^Device 1 (EtherCAT)^Term 1 (EK1200)^Term 11 (EK1122)^Term 12 (EK1100)^Term 24 (EK1322)^Box 4 (EPP2339-0021) X4^Channel 3^Input'}
bSens4s04D3 AT%I* :BOOL;	// Датчик сканирования RFID
{attribute 'TcLinkTo' := 'TIID^Device 1 (EtherCAT)^Term 1 (EK1200)^Term 11 (EK1122)^Term 12 (EK1100)^Term 24 (EK1322)^Box 4 (EPP2339-0021) X4^Channel 4^Input'}
bSens4s05D1 AT%I* :BOOL;	// Датчик в конце секции (в прямом направлении)
{attribute 'TcLinkTo' := 'TIID^Device 1 (EtherCAT)^Term 1 (EK1200)^Term 11 (EK1122)^Term 12 (EK1100)^Term 24 (EK1322)^Box 4 (EPP2339-0021) X4^Channel 5^Input'}
bSens4s05D2 AT%I* :BOOL;	// Датчик управления двойным движением
{attribute 'TcLinkTo' := 'TIID^Device 1 (EtherCAT)^Term 1 (EK1200)^Term 11 (EK1122)^Term 12 (EK1100)^Term 24 (EK1322)^Box 4 (EPP2339-0021) X4^Channel 6^Input'}
bSens4s06D1 AT%I* :BOOL;	// Датчик в конце секции (в прямом направлении)
{attribute 'TcLinkTo' := 'TIID^Device 1 (EtherCAT)^Term 1 (EK1200)^Term 11 (EK1122)^Term 12 (EK1100)^Term 24 (EK1322)^Box 4 (EPP2339-0021) X4^Channel 7^Input'}
bSens4s06D2 AT%I* :BOOL;	// Датчик контроля вил

END_VAR

// ---- GVLs/Conveyor_4/GVL_BusyFree_4.TcGVL
VAR_GLOBAL
(*Текущее состояние платформы (Занято/Свободно)*)
(*Первый этаж*)
	bPlatformBusy4s01	 	:BOOL;
	bPlatformFree4s01 		:BOOL;
	bPlatformBusy4s02 		:BOOL;
	bPlatformFree4s02 		:BOOL;
	bPlatformBusy4s03 		:BOOL;
	bPlatformFree4s03 		:BOOL;
	bPlatformBusy4s04 		:BOOL;
	bPlatformFree4s04 		:BOOL;
	bPlatformBusy4s05		:BOOL;
	bPlatformFree4s05 		:BOOL;
	bPlatformBusy4s06		:BOOL;
	bPlatformFree4s06 		:BOOL;
END_VAR

// ---- GVLs/Global_Variables.TcGVL

	VAR_GLOBAL CONSTANT
	PLCPRJ_BUFFER_SIZE						: UDINT := 1000;(* Max. internal fifo/receiver buffer size *)

(*	PLCPRJ_CLIENT_SEND_CYCLE_TIME			: TIME := T#1S; not used at server side *)
	PLCPRJ_RECEIVE_POLLING_TIME				: TIME := T#100MS;
	PLCPRJ_RECEIVE_TIMEOUT					: TIME := T#50S;

	(* Some project specific error codes *)
	PLCPRJ_ERROR_RECEIVE_TIMEOUT			: UDINT := 16#8101;(* Receive timeout *)
	PLCPRJ_ERROR_SENDFIFO_OVERFLOW			: UDINT := 16#8102;(* Send fifo overflow *)
	PLCPRJ_ERROR_RECFIFO_OVERFLOW			: UDINT := 16#8103;(* Receive fifo overflow *)
END_VAR

// ---- GVLs/GVL.TcGVL
VAR_GLOBAL

sSystemTime:STRING;

bAutomat1		  :BOOL;
bStartAutomat1	  :BOOL;
bManual1		  :BOOL;
bStop1			  :BOOL;
bReset1			  :BOOL := FALSE;
bDirect1		  :BOOL;
bReverse1		  :BOOL;
bBuffering1		  :BOOL:=TRUE;
//-------------------------//
bAutomat2		  :BOOL;
bStartAutomat2	  :BOOL;
bManual2		  :BOOL;
bStop2			  :BOOL;
bReset2			  :BOOL := FALSE;
bDirect2		  :BOOL;
bReverse2		  :BOOL;
bBuffering2		  :BOOL:=TRUE;
//-------------------------//
bAutomat3		  :BOOL;
bStartAutomat3	  :BOOL;
bManual3		  :BOOL;
bStop3			  :BOOL;
bReset3			  :BOOL := FALSE;
bDirect3		  :BOOL;
bReverse3		  :BOOL;
bBuffering3		  :BOOL:=TRUE;
//-------------------------//
bAutomat4		  :BOOL;
bStartAutomat4	  :BOOL;
bManual4		  :BOOL;
bStop4			  :BOOL;
bReset4			  :BOOL := FALSE;
bDirect4		  :BOOL;
bReverse4		  :BOOL;
bBuffering4		  :BOOL:=TRUE;
//-------------------------//

bSound1			  :BOOL;
bSound1_		  :BOOL;
bSound2			  :BOOL;
bSound2_		  :BOOL;
bSound3			  :BOOL;
bSound3_		  :BOOL;
bSound4			  :BOOL;
bSound4_		  :BOOL;

blink			  :BLINK;
Out1 		AT%Q* :BOOL;   //Выход на дискретный вход RFID Alien

{attribute 'TcLinkTo' := 'TIID^Device 1 (EtherCAT)^Term 1 (EK1200)^Term 13 (EK1322)^Box 1 (EPP2339-0021) X1^Channel 25^Output'}
b_1S4_2A2  AT%Q*  :BOOL;   // ALR F800 приемник RFID 1 (RFID scan)
{attribute 'TcLinkTo' := 'TIID^Device 1 (EtherCAT)^Term 1 (EK1200)^Term 13 (EK1322)^Box 4 (EPP2339-0021) X2^Channel 25^Output'}
b_2S4_2A2  AT%Q*  :BOOL;   // ALR F800 приемник RFID 2 (RFID scan)
{attribute 'TcLinkTo' := 'TIID^Device 1 (EtherCAT)^Term 1 (EK1200)^Term 11 (EK1122)^Term 12 (EK1100)^Term 24 (EK1322)^Box 1 (EPP2339-0021) X3^Channel 25^Output'}
b_3S4_2A2  AT%Q*  :BOOL;   // ALR F800 приемник RFID 3 (RFID scan)
{attribute 'TcLinkTo' := 'TIID^Device 1 (EtherCAT)^Term 1 (EK1200)^Term 11 (EK1122)^Term 12 (EK1100)^Term 24 (EK1322)^Box 4 (EPP2339-0021) X4^Channel 25^Output'}
b_4S4_2A2  AT%Q*  :BOOL;   // ALR F800 приемник RFID 4 (RFID scan)

RFID_ID_1 		  :STRING; // QR-code полученый с RFID 1
RFID_ID_2 		  :STRING; // QR-code полученый с RFID 2
RFID_ID_3 		  :STRING; // QR-code полученый с RFID 3
RFID_ID_4 		  :STRING; // QR-code полученый с RFID 4

{attribute 'TcLinkTo' := 'TIID^Device 1 (EtherCAT)^Term 1 (EK1200)^Term 13 (EK1322)^Box 1 (EPP2339-0021) X1^Channel 26^Output'}
b_1S5_2A1   AT%Q* :BOOL; // Bizerba WM-3 модуль логики весов 1
{attribute 'TcLinkTo' := 'TIID^Device 1 (EtherCAT)^Term 1 (EK1200)^Term 13 (EK1322)^Box 4 (EPP2339-0021) X2^Channel 26^Output'}
b_2S5_2A1   AT%Q* :BOOL; // Bizerba WM-3 модуль логики весов 2
{attribute 'TcLinkTo' := 'TIID^Device 1 (EtherCAT)^Term 1 (EK1200)^Term 11 (EK1122)^Term 12 (EK1100)^Term 24 (EK1322)^Box 1 (EPP2339-0021) X3^Channel 26^Output'}
b_3S5_2A1   AT%Q* :BOOL; // Bizerba WM-3 модуль логики весов 3
{attribute 'TcLinkTo' := 'TIID^Device 1 (EtherCAT)^Term 1 (EK1200)^Term 11 (EK1122)^Term 12 (EK1100)^Term 24 (EK1322)^Box 4 (EPP2339-0021) X4^Channel 26^Output'}
b_4S5_2A1   AT%Q* :BOOL; // Bizerba WM-3 модуль логики весов 4

{attribute 'TcLinkTo' := 'TIID^Device 2 (Profinet Controller CCAT (RT))^scale1^API^Term 18 (Input 2 word)^Subterm 21 (Input 2 word)^Inputs^Input'}
Massa_1	 	AT%I* :REAL; // масса полученая с весов 1
Massa_1_INT		  :INT;	 //Преобразованное значение массы 1 из REAL в INT
Massa_1_Gramms	  :DINT; //Преобразованное значение массы 1 из Кг в Граммы
{attribute 'TcLinkTo' := 'TIID^Device 2 (Profinet Controller CCAT (RT))^scale2^API^Term 102 (Input 2 word)^Subterm 114 (Input 2 word)^Inputs^Input'}
Massa_2		AT%I* :REAL; // масса полученая с весов 2
Massa_2_INT		  :INT;	 //Преобразованное значение массы 2 из REAL в INT
Massa_2_Gramms	  :DINT; //Преобразованное значение массы 2 из Кг в Граммы
{attribute 'TcLinkTo' := 'TIID^Device 2 (Profinet Controller CCAT (RT))^scale3^API^Term 48 (Input 2 word)^Subterm 60 (Input 2 word)^Inputs^Input'}
Massa_3		AT%I* :REAL; // масса полученая с весов 3
Massa_3_INT		  :INT;  //Преобразованное значение массы 3 из REAL в INT
Massa_3_Gramms	  :DINT; //Преобразованное значение массы 3 из Кг в Граммы
{attribute 'TcLinkTo' := 'TIID^Device 2 (Profinet Controller CCAT (RT))^scale4^API^Term 75 (Input 2 word)^Subterm 87 (Input 2 word)^Inputs^Input'}
Massa_4		AT%I* :REAL; // масса полученая с весов 4
Massa_4_INT		  :INT;	 //Преобразованное значение массы 4 из REAL в INT
Massa_4_Gramms	  :DINT; //Преобразованное значение массы 4 из Кг в Граммы

{attribute 'TcLinkTo' := 'TIID^Device 1 (EtherCAT)^Term 1 (EK1200)^Term 2 (EL1008)^Channel 1^Input'}
b_1QF		AT%I* :BOOL; // Состояние AB 1QF (Защита УЗИП)
{attribute 'TcLinkTo' := 'TIID^Device 1 (EtherCAT)^Term 1 (EK1200)^Term 2 (EL1008)^Channel 2^Input'}
b_2QF		AT%I* :BOOL; // Состояние AB 2QF (питание +2.ШУ)
{attribute 'TcLinkTo' := 'TIID^Device 1 (EtherCAT)^Term 1 (EK1200)^Term 2 (EL1008)^Channel 3^Input'}
b_SF3		AT%I* :BOOL; // Состояние AB SF3 (всп.системы +1.ШУ)
{attribute 'TcLinkTo' := 'TIID^Device 1 (EtherCAT)^Term 1 (EK1200)^Term 2 (EL1008)^Channel 4^Input'}
b_K2		AT%I* :BOOL; // Авария ввода -К2
{attribute 'TcLinkTo' := 'TIID^Device 1 (EtherCAT)^Term 1 (EK1200)^Term 2 (EL1008)^Channel 5^Input'}
b_1AS1		AT%I* :BOOL; // Реле безопасности конвейера 1 1AS1
{attribute 'TcLinkTo' := 'TIID^Device 1 (EtherCAT)^Term 1 (EK1200)^Term 2 (EL1008)^Channel 6^Input'}
b_2AS1		AT%I* :BOOL; // Реле безопасности конвейера 2 1AS2
{attribute 'TcLinkTo' := 'TIID^Device 1 (EtherCAT)^Term 1 (EK1200)^Term 2 (EL1008)^Channel 7^Input'}
b_GP3		AT%I* :BOOL; // Состояние БП24В GP3

{attribute 'TcLinkTo' := 'TIID^Device 1 (EtherCAT)^Term 1 (EK1200)^Term 3 (EL1008)^Channel 1^Input'}
b_1QF1		AT%I* :BOOL; // Состояние AB 1QF1 (питание приводов конв.1)
{attribute 'TcLinkTo' := 'TIID^Device 1 (EtherCAT)^Term 1 (EK1200)^Term 3 (EL1008)^Channel 2^Input'}
b_1KM1_1 	AT%I* :BOOL; // Состояние 1КМ1.1 (конв.1 прямое вращение)
{attribute 'TcLinkTo' := 'TIID^Device 1 (EtherCAT)^Term 1 (EK1200)^Term 3 (EL1008)^Channel 3^Input'}
b_1KM1_2 	AT%I* :BOOL; // Состояние 1КМ1.2 (конв.1 реверсивное вращение)
{attribute 'TcLinkTo' := 'TIID^Device 1 (EtherCAT)^Term 1 (EK1200)^Term 3 (EL1008)^Channel 4^Input'}
b_2QF1		AT%I* :BOOL; // Состояние AB 2QF1 (питание приводов конв.2)
{attribute 'TcLinkTo' := 'TIID^Device 1 (EtherCAT)^Term 1 (EK1200)^Term 3 (EL1008)^Channel 5^Input'}
b_2KM1_1 	AT%I* :BOOL; // Состояние 2КМ1.1 (конв.2 прямое вращение)
{attribute 'TcLinkTo' := 'TIID^Device 1 (EtherCAT)^Term 1 (EK1200)^Term 3 (EL1008)^Channel 6^Input'}
b_2KM1_2 	AT%I* :BOOL; // Состояние 2КМ1.2 (конв.2 реверсивное вращение)
{attribute 'TcLinkTo' := 'TIID^Device 1 (EtherCAT)^Term 1 (EK1200)^Term 3 (EL1008)^Channel 7^Input'}
b_1P_I		AT%I* :BOOL; // Контроль превышения тока ввода
{attribute 'TcLinkTo' := 'TIID^Device 1 (EtherCAT)^Term 1 (EK1200)^Term 3 (EL1008)^Channel 8^Input'}
b_1P_U		AT%I* :BOOL; // Контроль превышения напряжения на вводе

{attribute 'TcLinkTo' := 'TIID^Device 1 (EtherCAT)^Term 1 (EK1200)^Term 4 (EL1008)^Channel 1^Input'}
b_1QF2_1QF7 AT%I* :BOOL; // Состояние AB 1QF2,1QF3,1QF4,1QF5,1QF6,1QF7 (питание привода конвейер 1 1М1)
{attribute 'TcLinkTo' := 'TIID^Device 1 (EtherCAT)^Term 1 (EK1200)^Term 4 (EL1008)^Channel 2^Input'}
b_1QF8		AT%I* :BOOL; // Состояние AB 1QF8 (питание тормозов конвейер 1)
{attribute 'TcLinkTo' := 'TIID^Device 1 (EtherCAT)^Term 1 (EK1200)^Term 4 (EL1008)^Channel 3^Input'}
b_1KM2		AT%I* :BOOL; // Состояние 1КМ2 (питание тормоза конвейер 1 1BR1)
{attribute 'TcLinkTo' := 'TIID^Device 1 (EtherCAT)^Term 1 (EK1200)^Term 4 (EL1008)^Channel 4^Input'}
b_1KM3		AT%I* :BOOL; // Состояние 1КМ3 (питание тормоза конвейер 1 1BR2)
{attribute 'TcLinkTo' := 'TIID^Device 1 (EtherCAT)^Term 1 (EK1200)^Term 4 (EL1008)^Channel 5^Input'}
b_1KM4		AT%I* :BOOL; // Состояние 1КМ4 (питание тормоза конвейер 1 1BR3)
{attribute 'TcLinkTo' := 'TIID^Device 1 (EtherCAT)^Term 1 (EK1200)^Term 4 (EL1008)^Channel 6^Input'}
b_1KM5		AT%I* :BOOL; // Состояние 1КМ5 (питание тормоза конвейер 1 1BR4)
{attribute 'TcLinkTo' := 'TIID^Device 1 (EtherCAT)^Term 1 (EK1200)^Term 4 (EL1008)^Channel 7^Input'}
b_1KM6		AT%I* :BOOL; // Состояние 1КМ6 (питание тормоза конвейер 1 1BR5)
{attribute 'TcLinkTo' := 'TIID^Device 1 (EtherCAT)^Term 1 (EK1200)^Term 4 (EL1008)^Channel 8^Input'}
b_1KM7		AT%I* :BOOL; // Состояние 1КМ7 (питание тормоза конвейер 1 1BR6)

{attribute 'TcLinkTo' := 'TIID^Device 1 (EtherCAT)^Term 1 (EK1200)^Term 5 (EL1008)^Channel 1^Input'}
b_2QF2_2QF7 AT%I* :BOOL; // Состояние AB 2QF2,2QF3,2QF4,2QF5,2QF6,2QF7 (питание привода конвейер 2 2М1)
{attribute 'TcLinkTo' := 'TIID^Device 1 (EtherCAT)^Term 1 (EK1200)^Term 5 (EL1008)^Channel 2^Input'}
b_2QF8		AT%I* :BOOL; // Состояние AB 2QF8 (питание тормозов конвейер 2)
{attribute 'TcLinkTo' := 'TIID^Device 1 (EtherCAT)^Term 1 (EK1200)^Term 5 (EL1008)^Channel 3^Input'}
b_2KM2		AT%I* :BOOL; // Состояние 2КМ2 (питание тормоза конвейер 2 2BR1)
{attribute 'TcLinkTo' := 'TIID^Device 1 (EtherCAT)^Term 1 (EK1200)^Term 5 (EL1008)^Channel 4^Input'}
b_2KM3		AT%I* :BOOL; // Состояние 2КМ3 (питание тормоза конвейер 2 2BR2)
{attribute 'TcLinkTo' := 'TIID^Device 1 (EtherCAT)^Term 1 (EK1200)^Term 5 (EL1008)^Channel 5^Input'}
b_2KM4		AT%I* :BOOL; // Состояние 2КМ4 (питание тормоза конвейер 2 2BR3)
{attribute 'TcLinkTo' := 'TIID^Device 1 (EtherCAT)^Term 1 (EK1200)^Term 5 (EL1008)^Channel 6^Input'}
b_2KM5		AT%I* :BOOL; // Состояние 2КМ5 (питание тормоза конвейер 2 2BR4)
{attribute 'TcLinkTo' := 'TIID^Device 1 (EtherCAT)^Term 1 (EK1200)^Term 5 (EL1008)^Channel 7^Input'}
b_2KM6		AT%I* :BOOL; // Состояние 2КМ6 (питание тормоза конвейер 2 2BR5)
{attribute 'TcLinkTo' := 'TIID^Device 1 (EtherCAT)^Term 1 (EK1200)^Term 5 (EL1008)^Channel 8^Input'}
b_2KM7		AT%I* :BOOL; // Состояние 2КМ7 (питание тормоза конвейер 2 2BR6)

{attribute 'TcLinkTo' := 'TIID^Device 1 (EtherCAT)^Term 1 (EK1200)^Term 7 (EL2008)^Channel 1^Output'}
b_1K1_1		AT%Q* :BOOL; // Включение 1КМ1.1
{attribute 'TcLinkTo' := 'TIID^Device 1 (EtherCAT)^Term 1 (EK1200)^Term 7 (EL2008)^Channel 2^Output'}
b_1K1_2		AT%Q* :BOOL; // Включение 1КМ1.2
{attribute 'TcLinkTo' := 'TIID^Device 1 (EtherCAT)^Term 1 (EK1200)^Term 7 (EL2008)^Channel 3^Output'}
b_2K1_1		AT%Q* :BOOL; // Включение 2КМ1.1
{attribute 'TcLinkTo' := 'TIID^Device 1 (EtherCAT)^Term 1 (EK1200)^Term 7 (EL2008)^Channel 4^Output'}
b_2K1_2		AT%Q* :BOOL; // Включение 2КМ1.2
{attribute 'TcLinkTo' := 'TIID^Device 1 (EtherCAT)^Term 1 (EK1200)^Term 7 (EL2008)^Channel 5^Output'}
b1K2		AT%Q* :BOOL; // Пуск 1UZ1
{attribute 'TcLinkTo' := 'TIID^Device 1 (EtherCAT)^Term 1 (EK1200)^Term 7 (EL2008)^Channel 6^Output'}
b1K3		AT%Q* :BOOL; // Пуск 1UZ2
{attribute 'TcLinkTo' := 'TIID^Device 1 (EtherCAT)^Term 1 (EK1200)^Term 7 (EL2008)^Channel 7^Output'}
b1K4		AT%Q* :BOOL; // Пуск 1UZ3
{attribute 'TcLinkTo' := 'TIID^Device 1 (EtherCAT)^Term 1 (EK1200)^Term 7 (EL2008)^Channel 8^Output'}
b1K5		AT%Q* :BOOL; // Пуск 1UZ4

{attribute 'TcLinkTo' := 'TIID^Device 1 (EtherCAT)^Term 1 (EK1200)^Term 8 (EL2008)^Channel 1^Output'}
b1K6		AT%Q* :BOOL; // Пуск 1UZ5
{attribute 'TcLinkTo' := 'TIID^Device 1 (EtherCAT)^Term 1 (EK1200)^Term 8 (EL2008)^Channel 2^Output'}
b1K7		AT%Q* :BOOL; // Пуск 1UZ6
{attribute 'TcLinkTo' := 'TIID^Device 1 (EtherCAT)^Term 1 (EK1200)^Term 8 (EL2008)^Channel 3^Output'}
b2K2		AT%Q* :BOOL; // Пуск 2UZ1
{attribute 'TcLinkTo' := 'TIID^Device 1 (EtherCAT)^Term 1 (EK1200)^Term 8 (EL2008)^Channel 4^Output'}
b2K3		AT%Q* :BOOL; // Пуск 2UZ2
{attribute 'TcLinkTo' := 'TIID^Device 1 (EtherCAT)^Term 1 (EK1200)^Term 8 (EL2008)^Channel 5^Output'}
b2K4		AT%Q* :BOOL; // Пуск 2UZ3
{attribute 'TcLinkTo' := 'TIID^Device 1 (EtherCAT)^Term 1 (EK1200)^Term 8 (EL2008)^Channel 6^Output'}
b2K5		AT%Q* :BOOL; // Пуск 2UZ4
{attribute 'TcLinkTo' := 'TIID^Device 1 (EtherCAT)^Term 1 (EK1200)^Term 8 (EL2008)^Channel 7^Output'}
b2K6		AT%Q* :BOOL; // Пуск 2UZ5
{attribute 'TcLinkTo' := 'TIID^Device 1 (EtherCAT)^Term 1 (EK1200)^Term 8 (EL2008)^Channel 8^Output'}
b2K7		AT%Q* :BOOL; // Пуск 2UZ6

{attribute 'TcLinkTo' := 'TIID^Device 1 (EtherCAT)^Term 1 (EK1200)^Term 13 (EK1322)^Box 3 (EPP2339-0021) X1^Channel 9^Input'}
b1_S1_SB0	AT%I* :BOOL; // Кнопка аварийного останова на стойке стеллажа 1
{attribute 'TcLinkTo' := 'TIID^Device 1 (EtherCAT)^Term 1 (EK1200)^Term 13 (EK1322)^Box 1 (EPP2339-0021) X1^Channel 11^Input'}
b1_S6_SB0	AT%I* :BOOL; // Кнопка аварийного останова 1
{attribute 'TcLinkTo' := 'TIID^Device 1 (EtherCAT)^Term 1 (EK1200)^Term 13 (EK1322)^Box 6 (EPP2339-0021) X2^Channel 9^Input'}
b2_S1_SB0	AT%I* :BOOL; // Кнопка аварийного останова на стойке стеллажа 2
{attribute 'TcLinkTo' := 'TIID^Device 1 (EtherCAT)^Term 1 (EK1200)^Term 13 (EK1322)^Box 4 (EPP2339-0021) X2^Channel 11^Input'}
b2_S6_SB0	AT%I* :BOOL; // Кнопка аварийного останова 2
{attribute 'TcLinkTo' := 'TIID^Device 1 (EtherCAT)^Term 1 (EK1200)^Term 11 (EK1122)^Term 12 (EK1100)^Term 24 (EK1322)^Box 3 (EPP2339-0021) X3^Channel 9^Input'}
b3_S1_SB0	AT%I* :BOOL; // Кнопка аварийного останова на стойке стеллажа 3
{attribute 'TcLinkTo' := 'TIID^Device 1 (EtherCAT)^Term 1 (EK1200)^Term 11 (EK1122)^Term 12 (EK1100)^Term 24 (EK1322)^Box 1 (EPP2339-0021) X3^Channel 11^Input'}
b3_S6_SB0	AT%I* :BOOL; // Кнопка аварийного останова 3
{attribute 'TcLinkTo' := 'TIID^Device 1 (EtherCAT)^Term 1 (EK1200)^Term 11 (EK1122)^Term 12 (EK1100)^Term 24 (EK1322)^Box 6 (EPP2339-0021) X4^Channel 9^Input'}
b4_S1_SB0	AT%I* :BOOL; // Кнопка аварийного останова на стойке стеллажа 4
{attribute 'TcLinkTo' := 'TIID^Device 1 (EtherCAT)^Term 1 (EK1200)^Term 11 (EK1122)^Term 12 (EK1100)^Term 24 (EK1322)^Box 4 (EPP2339-0021) X4^Channel 11^Input'}
b4_S6_SB0	AT%I* :BOOL; // Кнопка аварийного останова 4


{attribute 'TcLinkTo' := 'TIID^Device 1 (EtherCAT)^Term 1 (EK1200)^Term 9 (EL2008)^Channel 1^Output'}
b1S1_SB0	AT%Q* :BOOL; // Лампа SB0 +1.S1-SB0
{attribute 'TcLinkTo' := 'TIID^Device 1 (EtherCAT)^Term 1 (EK1200)^Term 9 (EL2008)^Channel 2^Output'}
b1S6_SB0	AT%Q* :BOOL; // Лампа SB0 +1.S6-SB0
{attribute 'TcLinkTo' := 'TIID^Device 1 (EtherCAT)^Term 1 (EK1200)^Term 9 (EL2008)^Channel 3^Output'}
b2S1_SB0	AT%Q* :BOOL; // Лампа SB0 +2.S1-SB0
{attribute 'TcLinkTo' := 'TIID^Device 1 (EtherCAT)^Term 1 (EK1200)^Term 9 (EL2008)^Channel 4^Output'}
b2S6_SB0	AT%Q* :BOOL; // Лампа SB0 +2.S6-SB0
{attribute 'TcLinkTo' := 'TIID^Device 1 (EtherCAT)^Term 1 (EK1200)^Term 9 (EL2008)^Channel 5^Output'}
b1Sh_SB0	AT%Q* :BOOL; // Лампа SB0 +1ШУ-1SB0
{attribute 'TcLinkTo' := 'TIID^Device 1 (EtherCAT)^Term 1 (EK1200)^Term 9 (EL2008)^Channel 6^Output'}
b1Sh_SB1	AT%Q* :BOOL; // Лампа Рестарт +1ШУ-1SB1

//-------------------------------------------------------------------------------------//

{attribute 'TcLinkTo' := 'TIID^Device 1 (EtherCAT)^Term 1 (EK1200)^Term 11 (EK1122)^Term 12 (EK1100)^Term 15 (EL1008)^Channel 1^Input'}
b_SF3_		AT%I* :BOOL; // Состояние AB SF3 (всп.системы +1.ШУ)
{attribute 'TcLinkTo' := 'TIID^Device 1 (EtherCAT)^Term 1 (EK1200)^Term 11 (EK1122)^Term 12 (EK1100)^Term 15 (EL1008)^Channel 2^Input'}
b_K2_		AT%I* :BOOL; // Авария ввода -К2
{attribute 'TcLinkTo' := 'TIID^Device 1 (EtherCAT)^Term 1 (EK1200)^Term 11 (EK1122)^Term 12 (EK1100)^Term 15 (EL1008)^Channel 3^Input'}
b_3AS1		AT%I* :BOOL; // Реле безопасности конвейера 3 3AS1
{attribute 'TcLinkTo' := 'TIID^Device 1 (EtherCAT)^Term 1 (EK1200)^Term 11 (EK1122)^Term 12 (EK1100)^Term 15 (EL1008)^Channel 4^Input'}
b_4AS1		AT%I* :BOOL; // Реле безопасности конвейера 4 4AS2

{attribute 'TcLinkTo' := 'TIID^Device 1 (EtherCAT)^Term 1 (EK1200)^Term 11 (EK1122)^Term 12 (EK1100)^Term 16 (EL1008)^Channel 1^Input'}
b_3QF1		AT%I* :BOOL; // Состояние AB 3QF1 (питание приводов конв.3)
{attribute 'TcLinkTo' := 'TIID^Device 1 (EtherCAT)^Term 1 (EK1200)^Term 11 (EK1122)^Term 12 (EK1100)^Term 16 (EL1008)^Channel 2^Input'}
b_3KM1_1	AT%I* :BOOL; // Состояние 3КМ1.1 (конв.3 прямое вращение)
{attribute 'TcLinkTo' := 'TIID^Device 1 (EtherCAT)^Term 1 (EK1200)^Term 11 (EK1122)^Term 12 (EK1100)^Term 16 (EL1008)^Channel 3^Input'}
b_3KM1_2	AT%I* :BOOL; // Состояние 3КМ1.2 (конв.3 реверсивное вращение)
{attribute 'TcLinkTo' := 'TIID^Device 1 (EtherCAT)^Term 1 (EK1200)^Term 11 (EK1122)^Term 12 (EK1100)^Term 16 (EL1008)^Channel 4^Input'}
b_4QF1		AT%I* :BOOL; // Состояние AB 4QF1 (питание приводов конв.4)
{attribute 'TcLinkTo' := 'TIID^Device 1 (EtherCAT)^Term 1 (EK1200)^Term 11 (EK1122)^Term 12 (EK1100)^Term 16 (EL1008)^Channel 5^Input'}
b_4KM1_1	AT%I* :BOOL; // Состояние 4КМ1.1 (конв.4 прямое вращение)
{attribute 'TcLinkTo' := 'TIID^Device 1 (EtherCAT)^Term 1 (EK1200)^Term 11 (EK1122)^Term 12 (EK1100)^Term 16 (EL1008)^Channel 6^Input'}
b_4KM1_2	AT%I* :BOOL; // Состояние 4КМ1.2 (конв.4 реверсивное вращение)

{attribute 'TcLinkTo' := 'TIID^Device 1 (EtherCAT)^Term 1 (EK1200)^Term 11 (EK1122)^Term 12 (EK1100)^Term 17 (EL1008)^Channel 1^Input'}
b_3QF2_3QF7 AT%I* :BOOL; // Состояние AB 3QF2,3QF3,3QF4,3QF5,3QF6,3QF7 (питание привода конвейер 3 1М1)
{attribute 'TcLinkTo' := 'TIID^Device 1 (EtherCAT)^Term 1 (EK1200)^Term 11 (EK1122)^Term 12 (EK1100)^Term 17 (EL1008)^Channel 2^Input'}
b_3QF8		AT%I* :BOOL; // Состояние AB 3QF8 (питание тормозов конвейер 3)
{attribute 'TcLinkTo' := 'TIID^Device 1 (EtherCAT)^Term 1 (EK1200)^Term 11 (EK1122)^Term 12 (EK1100)^Term 17 (EL1008)^Channel 3^Input'}
b_3KM2		AT%I* :BOOL; // Состояние 3КМ2 (питание тормоза конвейер 3 3BR1)
{attribute 'TcLinkTo' := 'TIID^Device 1 (EtherCAT)^Term 1 (EK1200)^Term 11 (EK1122)^Term 12 (EK1100)^Term 17 (EL1008)^Channel 4^Input'}
b_3KM3		AT%I* :BOOL; // Состояние 3КМ3 (питание тормоза конвейер 3 3BR2)
{attribute 'TcLinkTo' := 'TIID^Device 1 (EtherCAT)^Term 1 (EK1200)^Term 11 (EK1122)^Term 12 (EK1100)^Term 17 (EL1008)^Channel 5^Input'}
b_3KM4		AT%I* :BOOL; // Состояние 3КМ4 (питание тормоза конвейер 3 3BR3)
{attribute 'TcLinkTo' := 'TIID^Device 1 (EtherCAT)^Term 1 (EK1200)^Term 11 (EK1122)^Term 12 (EK1100)^Term 17 (EL1008)^Channel 6^Input'}
b_3KM5		AT%I* :BOOL; // Состояние 3КМ5 (питание тормоза конвейер 3 3BR4)
{attribute 'TcLinkTo' := 'TIID^Device 1 (EtherCAT)^Term 1 (EK1200)^Term 11 (EK1122)^Term 12 (EK1100)^Term 17 (EL1008)^Channel 7^Input'}
b_3KM6		AT%I* :BOOL; // Состояние 3КМ6 (питание тормоза конвейер 3 3BR5)
{attribute 'TcLinkTo' := 'TIID^Device 1 (EtherCAT)^Term 1 (EK1200)^Term 11 (EK1122)^Term 12 (EK1100)^Term 17 (EL1008)^Channel 8^Input'}
b_3KM7		AT%I* :BOOL; // Состояние 3КМ7 (питание тормоза конвейер 3 3BR6)

{attribute 'TcLinkTo' := 'TIID^Device 1 (EtherCAT)^Term 1 (EK1200)^Term 11 (EK1122)^Term 12 (EK1100)^Term 18 (EL1008)^Channel 1^Input'}
b_4QF2_4QF7 AT%I* :BOOL; // Состояние AB 4QF2,4QF3,4QF4,4QF5,4QF6,4QF7 (питание привода конвейер 4 2М1)
{attribute 'TcLinkTo' := 'TIID^Device 1 (EtherCAT)^Term 1 (EK1200)^Term 11 (EK1122)^Term 12 (EK1100)^Term 18 (EL1008)^Channel 2^Input'}
b_4QF8		AT%I* :BOOL; // Состояние AB 4QF8 (питание тормозов конвейер 4)
{attribute 'TcLinkTo' := 'TIID^Device 1 (EtherCAT)^Term 1 (EK1200)^Term 11 (EK1122)^Term 12 (EK1100)^Term 18 (EL1008)^Channel 3^Input'}
b_4KM2		AT%I* :BOOL; // Состояние 4КМ2 (питание тормоза конвейер 4 4BR1)
{attribute 'TcLinkTo' := 'TIID^Device 1 (EtherCAT)^Term 1 (EK1200)^Term 11 (EK1122)^Term 12 (EK1100)^Term 18 (EL1008)^Channel 4^Input'}
b_4KM3		AT%I* :BOOL; // Состояние 4КМ3 (питание тормоза конвейер 4 4BR2)
{attribute 'TcLinkTo' := 'TIID^Device 1 (EtherCAT)^Term 1 (EK1200)^Term 11 (EK1122)^Term 12 (EK1100)^Term 18 (EL1008)^Channel 5^Input'}
b_4KM4		AT%I* :BOOL; // Состояние 4КМ4 (питание тормоза конвейер 4 4BR3)
{attribute 'TcLinkTo' := 'TIID^Device 1 (EtherCAT)^Term 1 (EK1200)^Term 11 (EK1122)^Term 12 (EK1100)^Term 18 (EL1008)^Channel 6^Input'}
b_4KM5		AT%I* :BOOL; // Состояние 4КМ5 (питание тормоза конвейер 4 4BR4)
{attribute 'TcLinkTo' := 'TIID^Device 1 (EtherCAT)^Term 1 (EK1200)^Term 11 (EK1122)^Term 12 (EK1100)^Term 18 (EL1008)^Channel 7^Input'}
b_4KM6		AT%I* :BOOL; // Состояние 4КМ6 (питание тормоза конвейер 4 4BR5)
{attribute 'TcLinkTo' := 'TIID^Device 1 (EtherCAT)^Term 1 (EK1200)^Term 11 (EK1122)^Term 12 (EK1100)^Term 18 (EL1008)^Channel 8^Input'}
b_4KM7		AT%I* :BOOL; // Состояние 4КМ7 (питание тормоза конвейер 4 4BR6)

{attribute 'TcLinkTo' := 'TIID^Device 1 (EtherCAT)^Term 1 (EK1200)^Term 11 (EK1122)^Term 12 (EK1100)^Term 20 (EL2008)^Channel 1^Output'}
b_3K1_1		AT%Q* :BOOL; // Включение 3КМ1.1
{attribute 'TcLinkTo' := 'TIID^Device 1 (EtherCAT)^Term 1 (EK1200)^Term 11 (EK1122)^Term 12 (EK1100)^Term 20 (EL2008)^Channel 2^Output'}
b_3K1_2		AT%Q* :BOOL; // Включение 3КМ1.2
{attribute 'TcLinkTo' := 'TIID^Device 1 (EtherCAT)^Term 1 (EK1200)^Term 11 (EK1122)^Term 12 (EK1100)^Term 20 (EL2008)^Channel 3^Output'}
b_4K1_1		AT%Q* :BOOL; // Включение 4КМ1.1
{attribute 'TcLinkTo' := 'TIID^Device 1 (EtherCAT)^Term 1 (EK1200)^Term 11 (EK1122)^Term 12 (EK1100)^Term 20 (EL2008)^Channel 4^Output'}
b_4K1_2		AT%Q* :BOOL; // Включение 4КМ1.2
{attribute 'TcLinkTo' := 'TIID^Device 1 (EtherCAT)^Term 1 (EK1200)^Term 11 (EK1122)^Term 12 (EK1100)^Term 20 (EL2008)^Channel 5^Output'}
b3K2		AT%Q* :BOOL; // Пуск 3UZ1
{attribute 'TcLinkTo' := 'TIID^Device 1 (EtherCAT)^Term 1 (EK1200)^Term 11 (EK1122)^Term 12 (EK1100)^Term 20 (EL2008)^Channel 6^Output'}
b3K3		AT%Q* :BOOL; // Пуск 3UZ2
{attribute 'TcLinkTo' := 'TIID^Device 1 (EtherCAT)^Term 1 (EK1200)^Term 11 (EK1122)^Term 12 (EK1100)^Term 20 (EL2008)^Channel 7^Output'}
b3K4		AT%Q* :BOOL; // Пуск 3UZ3
{attribute 'TcLinkTo' := 'TIID^Device 1 (EtherCAT)^Term 1 (EK1200)^Term 11 (EK1122)^Term 12 (EK1100)^Term 20 (EL2008)^Channel 8^Output'}
b3K5		AT%Q* :BOOL; // Пуск 3UZ4

{attribute 'TcLinkTo' := 'TIID^Device 1 (EtherCAT)^Term 1 (EK1200)^Term 11 (EK1122)^Term 12 (EK1100)^Term 21 (EL2008)^Channel 1^Output'}
b3K6		AT%Q* :BOOL; // Пуск 3UZ5
{attribute 'TcLinkTo' := 'TIID^Device 1 (EtherCAT)^Term 1 (EK1200)^Term 11 (EK1122)^Term 12 (EK1100)^Term 21 (EL2008)^Channel 2^Output'}
b3K7		AT%Q* :BOOL; // Пуск 3UZ6
{attribute 'TcLinkTo' := 'TIID^Device 1 (EtherCAT)^Term 1 (EK1200)^Term 11 (EK1122)^Term 12 (EK1100)^Term 21 (EL2008)^Channel 3^Output'}
b4K2		AT%Q* :BOOL; // Пуск 4UZ1
{attribute 'TcLinkTo' := 'TIID^Device 1 (EtherCAT)^Term 1 (EK1200)^Term 11 (EK1122)^Term 12 (EK1100)^Term 21 (EL2008)^Channel 4^Output'}
b4K3		AT%Q* :BOOL; // Пуск 4UZ2
{attribute 'TcLinkTo' := 'TIID^Device 1 (EtherCAT)^Term 1 (EK1200)^Term 11 (EK1122)^Term 12 (EK1100)^Term 21 (EL2008)^Channel 5^Output'}
b4K4		AT%Q* :BOOL; // Пуск 4UZ3
{attribute 'TcLinkTo' := 'TIID^Device 1 (EtherCAT)^Term 1 (EK1200)^Term 11 (EK1122)^Term 12 (EK1100)^Term 21 (EL2008)^Channel 6^Output'}
b4K5		AT%Q* :BOOL; // Пуск 4UZ4
{attribute 'TcLinkTo' := 'TIID^Device 1 (EtherCAT)^Term 1 (EK1200)^Term 11 (EK1122)^Term 12 (EK1100)^Term 21 (EL2008)^Channel 7^Output'}
b4K6		AT%Q* :BOOL; // Пуск 4UZ5
{attribute 'TcLinkTo' := 'TIID^Device 1 (EtherCAT)^Term 1 (EK1200)^Term 11 (EK1122)^Term 12 (EK1100)^Term 21 (EL2008)^Channel 8^Output'}
b4K7		AT%Q* :BOOL; // Пуск 4UZ6

{attribute 'TcLinkTo' := 'TIID^Device 1 (EtherCAT)^Term 1 (EK1200)^Term 11 (EK1122)^Term 12 (EK1100)^Term 22 (EL2008)^Channel 1^Output'}
b3S1_SB0	AT%Q* :BOOL; // Лампа SB0 +3.S1-SB0
{attribute 'TcLinkTo' := 'TIID^Device 1 (EtherCAT)^Term 1 (EK1200)^Term 11 (EK1122)^Term 12 (EK1100)^Term 22 (EL2008)^Channel 2^Output'}
b3S6_SB0	AT%Q* :BOOL; // Лампа SB0 +3.S6-SB0
{attribute 'TcLinkTo' := 'TIID^Device 1 (EtherCAT)^Term 1 (EK1200)^Term 11 (EK1122)^Term 12 (EK1100)^Term 22 (EL2008)^Channel 3^Output'}
b4S1_SB0	AT%Q* :BOOL; // Лампа SB0 +4.S1-SB0
{attribute 'TcLinkTo' := 'TIID^Device 1 (EtherCAT)^Term 1 (EK1200)^Term 11 (EK1122)^Term 12 (EK1100)^Term 22 (EL2008)^Channel 4^Output'}
b4S6_SB0	AT%Q* :BOOL; // Лампа SB0 +4.S6-SB0
{attribute 'TcLinkTo' := 'TIID^Device 1 (EtherCAT)^Term 1 (EK1200)^Term 11 (EK1122)^Term 12 (EK1100)^Term 22 (EL2008)^Channel 5^Output'}
b2Sh_SB0	AT%Q* :BOOL; // Лампа SB0 +2ШУ-1SB0
{attribute 'TcLinkTo' := 'TIID^Device 1 (EtherCAT)^Term 1 (EK1200)^Term 11 (EK1122)^Term 12 (EK1100)^Term 22 (EL2008)^Channel 6^Output'}
b2Sh_SB1	AT%Q* :BOOL; // Лампа Рестарт +2ШУ-1SB1

END_VAR

// ---- GVLs/GVL_Alarm.TcGVL
VAR_GLOBAL

	bNotReadyPower24v       	:BOOL;
	bPermAlarm1					:BOOL;

	bAlarm						:BOOL;
	bAlarm1						:BOOL;
	bAlarm1_vis					:BOOL; //Мигающая авария для визуализации конвейер 1
	bAlarm2						:BOOL;
	bAlarm2_vis					:BOOL; //Мигающая авария для визуализации конвейер 2
	bAlarm3						:BOOL;
	bAlarm3_vis					:BOOL; //Мигающая авария для визуализации конвейер 3
	bAlarm4						:BOOL;
	bAlarm4_vis					:BOOL; //Мигающая авария для визуализации конвейер 4
	
	bAlarm1QF					:BOOL;
	bAlarm2QF					:BOOL;

	bAlarmSF3					:BOOL;
	bAlarmSF3_					:BOOL;

	bAlarmK2					:BOOL;
	bAlarmK2_					:BOOL;

	bAlarm1AS1					:BOOL;
	bAlarm2AS1					:BOOL;
	bAlarm3AS1					:BOOL;
	bAlarm4AS1					:BOOL;

	bAlarm1QF1					:BOOL;
	bAlarm2QF1					:BOOL;
	bAlarm3QF1					:BOOL;
	bAlarm4QF1					:BOOL;

	bAlarm1P_I					:BOOL;
	bAlarm1P_U					:BOOL;

	bAlarm1QF2_1QF7				:BOOL;
	bAlarm1QF8					:BOOL;
	bAlarm1KM2					:BOOL;
	bAlarm1KM3					:BOOL;
	bAlarm1KM4					:BOOL;
	bAlarm1KM5					:BOOL;
	bAlarm1KM6					:BOOL;
	bAlarm1KM7					:BOOL;

	bAlarm2QF2_2QF7				:BOOL;	
	bAlarm2QF8					:BOOL;
	bAlarm2KM2					:BOOL;
	bAlarm2KM3					:BOOL;
	bAlarm2KM4					:BOOL;
	bAlarm2KM5					:BOOL;
	bAlarm2KM6					:BOOL;
	bAlarm2KM7					:BOOL;

	bAlarm3QF2_3QF7				:BOOL;
	bAlarm3QF8					:BOOL;
	bAlarm3KM2					:BOOL;
	bAlarm3KM3					:BOOL;
	bAlarm3KM4					:BOOL;
	bAlarm3KM5					:BOOL;
	bAlarm3KM6					:BOOL;
	bAlarm3KM7					:BOOL;

	bAlarm4QF2_4QF7				:BOOL;	
	bAlarm4QF8					:BOOL;
	bAlarm4KM2					:BOOL;
	bAlarm4KM3					:BOOL;
	bAlarm4KM4					:BOOL;
	bAlarm4KM5					:BOOL;
	bAlarm4KM6					:BOOL;
	bAlarm4KM7					:BOOL;
	
	bAlarm_b1_S1_SB0			:BOOL;
	bAlarm_b1_S6_SB0			:BOOL;
	bAlarm_b2_S1_SB0			:BOOL;
	bAlarm_b2_S6_SB0			:BOOL;
	bAlarm_b3_S1_SB0			:BOOL;
	bAlarm_b3_S6_SB0			:BOOL;
	bAlarm_b4_S1_SB0			:BOOL;
	bAlarm_b4_S6_SB0			:BOOL;
	
	bAlarmSafety1				:BOOL;
	bAlarmSafety2				:BOOL;
	bAlarmSafety3				:BOOL;
	bAlarmSafety4				:BOOL;
	
	bNotReady1					:BOOL;
	bNotReady2					:BOOL;
	bNotReady3					:BOOL;
	bNotReady4					:BOOL;
	
	bNotReady_1					:BOOL;
	bNotReady_2					:BOOL;
	bNotReady_3					:BOOL;
	bNotReady_4					:BOOL;
	
	bLongMove1					:BOOL;
	bLongMove2					:BOOL;
	bLongMove3					:BOOL;
	bLongMove4					:BOOL;
	
	bAlarmSF					:BOOL;
	bAlarm_input_accident		:BOOL;
	bAlarm_Safety_relay			:BOOL;
	bAlarm_Drive_power			:BOOL;
	bAlarmQF					:BOOL;
	bAlarm_Overload_I_U			:BOOL;

	bNotReadyGeneral			:BOOL;
	bNotReadyGeneral1			:BOOL;
	bNotReadyGeneral2			:BOOL;
	bNotReadyGeneral3			:BOOL;
	bNotReadyGeneral4			:BOOL;

	bAlarmGeneral				:BOOL;
	bAlarmGeneral1				:BOOL;
	bAlarmGeneral2				:BOOL;
	bAlarmGeneral3				:BOOL;
	bAlarmGeneral4				:BOOL;
	
	bButtAlarmResetHMI			:BOOL;
	bButtAlarmReset1 			:BOOL;
	bButtAlarmReset2 			:BOOL;
	bButtAlarmReset3 			:BOOL;
	bButtAlarmReset4 			:BOOL;

	bButtAlarmResetGeneral		:BOOL;	
	bButtAlarmResetGeneral1		:BOOL;
	bButtAlarmResetGeneral2		:BOOL;
	bButtAlarmResetGeneral3		:BOOL;
	bButtAlarmResetGeneral4		:BOOL;
	
	bAlarmResetGeneral			:BOOL;
	bAlarmReset1				:BOOL;
	bAlarmReset2				:BOOL;
	bAlarmReset3				:BOOL;
	bAlarmReset4				:BOOL;

	sAlarmLineGeneral			:WSTRING;	
	sAlarmLine1					:WSTRING;
	sAlarmLine2					:WSTRING;
	sAlarmLine3					:WSTRING;
	sAlarmLine4					:WSTRING;

	sAlarmGeneral				:WSTRING;
	sAlarm1						:WSTRING;
	sAlarm2						:WSTRING;
	sAlarm3						:WSTRING;
	sAlarm4						:WSTRING;
	
	bPermAlarmDrive1      		:BOOL;
	bPermAlarmDrive2      		:BOOL;
	bPermAlarmDrive3      		:BOOL;
	bPermAlarmDrive4      		:BOOL;
	
	bNotDriveReady1s01M1		:BOOL;
	bNotDriveReady1s02M1		:BOOL;
	bNotDriveReady1s03M1		:BOOL;
	bNotDriveReady1s04M1		:BOOL;
	bNotDriveReady1s05M1		:BOOL;
	bNotDriveReady1s06M1		:BOOL;
	
	bNotDriveReady2s01M1		:BOOL;
	bNotDriveReady2s02M1		:BOOL;
	bNotDriveReady2s03M1		:BOOL;
	bNotDriveReady2s04M1		:BOOL;
	bNotDriveReady2s05M1		:BOOL;
	bNotDriveReady2s06M1		:BOOL;
	
	bNotDriveReady3s01M1		:BOOL;
	bNotDriveReady3s02M1		:BOOL;
	bNotDriveReady3s03M1		:BOOL;
	bNotDriveReady3s04M1		:BOOL;
	bNotDriveReady3s05M1		:BOOL;
	bNotDriveReady3s06M1		:BOOL;

	bNotDriveReady4s01M1		:BOOL;
	bNotDriveReady4s02M1		:BOOL;
	bNotDriveReady4s03M1		:BOOL;
	bNotDriveReady4s04M1		:BOOL;
	bNotDriveReady4s05M1		:BOOL;
	bNotDriveReady4s06M1		:BOOL;
	
	b1K2_b1KM2_good 			:BOOL;
	b1K2_b1KM2_bad				:BOOL;
	b1K2_b1KM2_err				:BOOL;

	b1K3_b1KM3_good 			:BOOL;
	b1K3_b1KM3_bad				:BOOL;
	b1K3_b1KM3_err				:BOOL;

	b1K4_b1KM4_good 			:BOOL;
	b1K4_b1KM4_bad				:BOOL;
	b1K4_b1KM4_err				:BOOL;

	b1K5_b1KM5_good 			:BOOL;
	b1K5_b1KM5_bad				:BOOL;
	b1K5_b1KM5_err				:BOOL;

	b1K6_b1KM6_good 			:BOOL;
	b1K6_b1KM6_bad				:BOOL;
	b1K6_b1KM6_err				:BOOL;

	b1K7_b1KM7_good 			:BOOL;
	b1K7_b1KM7_bad				:BOOL;
	b1K7_b1KM7_err				:BOOL;

END_VAR

// ---- GVLs/GVL_Lights.TcGVL
VAR_GLOBAL
// Светофоры
// 4 цвета + сирена на стойке стеллажа h=3000мм Конвейер 1
{attribute 'TcLinkTo' := 'TIID^Device 1 (EtherCAT)^Term 1 (EK1200)^Term 13 (EK1322)^Box 1 (EPP2339-0021) X1^Channel 29^Output'}
	bRed_1S1HL1 			AT%Q*	:BOOL;
{attribute 'TcLinkTo' := 'TIID^Device 1 (EtherCAT)^Term 1 (EK1200)^Term 13 (EK1322)^Box 1 (EPP2339-0021) X1^Channel 30^Output'}
	bGreen_1S1HL1 			AT%Q*	:BOOL;
{attribute 'TcLinkTo' := 'TIID^Device 1 (EtherCAT)^Term 1 (EK1200)^Term 13 (EK1322)^Box 1 (EPP2339-0021) X1^Channel 31^Output'}
	bYellow_1S1HL1 	 		AT%Q*	:BOOL;
{attribute 'TcLinkTo' := 'TIID^Device 1 (EtherCAT)^Term 1 (EK1200)^Term 13 (EK1322)^Box 1 (EPP2339-0021) X1^Channel 32^Output'}
	bBlue_1S1HL1 			AT%Q*	:BOOL;
{attribute 'TcLinkTo' := 'TIID^Device 1 (EtherCAT)^Term 1 (EK1200)^Term 13 (EK1322)^Box 1 (EPP2339-0021) X1^Channel 28^Output'}
	bSound_1S1HL1			AT%Q*	:BOOL;
//---------------------------------------------------------------------------------------------------------------//
// 4 цвета + сирена на стойке стеллажа h=3000мм Конвейер 1
{attribute 'TcLinkTo' := 'TIID^Device 1 (EtherCAT)^Term 1 (EK1200)^Term 13 (EK1322)^Box 3 (EPP2339-0021) X1^Channel 21^Output'}
	bRed_1S1_HL1 			AT%Q*	:BOOL;
{attribute 'TcLinkTo' := 'TIID^Device 1 (EtherCAT)^Term 1 (EK1200)^Term 13 (EK1322)^Box 3 (EPP2339-0021) X1^Channel 22^Output'}
	bGreen_1S1_HL1 			AT%Q*	:BOOL;
{attribute 'TcLinkTo' := 'TIID^Device 1 (EtherCAT)^Term 1 (EK1200)^Term 13 (EK1322)^Box 3 (EPP2339-0021) X1^Channel 23^Output'}
	bYellow_1S1_HL1 	 	AT%Q*	:BOOL;
{attribute 'TcLinkTo' := 'TIID^Device 1 (EtherCAT)^Term 1 (EK1200)^Term 13 (EK1322)^Box 3 (EPP2339-0021) X1^Channel 24^Output'}
	bBlue_1S1_HL1 			AT%Q*	:BOOL;
{attribute 'TcLinkTo' := 'TIID^Device 1 (EtherCAT)^Term 1 (EK1200)^Term 13 (EK1322)^Box 3 (EPP2339-0021) X1^Channel 20^Output'}
	bSound_1S1_HL1			AT%Q*	:BOOL;
//---------------------------------------------------------------------------------------------------------------//
// 4 цвета + сирена на стойке стеллажа h=3000мм Конвейер 2
{attribute 'TcLinkTo' := 'TIID^Device 1 (EtherCAT)^Term 1 (EK1200)^Term 13 (EK1322)^Box 4 (EPP2339-0021) X2^Channel 29^Output'}
	bRed_2S1HL1 			AT%Q*	:BOOL;
{attribute 'TcLinkTo' := 'TIID^Device 1 (EtherCAT)^Term 1 (EK1200)^Term 13 (EK1322)^Box 4 (EPP2339-0021) X2^Channel 30^Output'}
	bGreen_2S1HL1 			AT%Q*	:BOOL;
{attribute 'TcLinkTo' := 'TIID^Device 1 (EtherCAT)^Term 1 (EK1200)^Term 13 (EK1322)^Box 4 (EPP2339-0021) X2^Channel 31^Output'}
	bYellow_2S1HL1 	 		AT%Q*	:BOOL;
{attribute 'TcLinkTo' := 'TIID^Device 1 (EtherCAT)^Term 1 (EK1200)^Term 13 (EK1322)^Box 4 (EPP2339-0021) X2^Channel 32^Output'}
	bBlue_2S1HL1 			AT%Q*	:BOOL;
{attribute 'TcLinkTo' := 'TIID^Device 1 (EtherCAT)^Term 1 (EK1200)^Term 13 (EK1322)^Box 4 (EPP2339-0021) X2^Channel 28^Output'}
	bSound_2S1HL1			AT%Q*	:BOOL;
//---------------------------------------------------------------------------------------------------------------//
// 4 цвета + сирена на стойке стеллажа h=3000мм Конвейер 2
{attribute 'TcLinkTo' := 'TIID^Device 1 (EtherCAT)^Term 1 (EK1200)^Term 13 (EK1322)^Box 6 (EPP2339-0021) X2^Channel 21^Output'}
	bRed_2S1_HL1 			AT%Q*	:BOOL;
{attribute 'TcLinkTo' := 'TIID^Device 1 (EtherCAT)^Term 1 (EK1200)^Term 13 (EK1322)^Box 6 (EPP2339-0021) X2^Channel 22^Output'}
	bGreen_2S1_HL1 			AT%Q*	:BOOL;
{attribute 'TcLinkTo' := 'TIID^Device 1 (EtherCAT)^Term 1 (EK1200)^Term 13 (EK1322)^Box 6 (EPP2339-0021) X2^Channel 23^Output'}
	bYellow_2S1_HL1 	 	AT%Q*	:BOOL;
{attribute 'TcLinkTo' := 'TIID^Device 1 (EtherCAT)^Term 1 (EK1200)^Term 13 (EK1322)^Box 6 (EPP2339-0021) X2^Channel 24^Output'}
	bBlue_2S1_HL1 			AT%Q*	:BOOL;
{attribute 'TcLinkTo' := 'TIID^Device 1 (EtherCAT)^Term 1 (EK1200)^Term 13 (EK1322)^Box 6 (EPP2339-0021) X2^Channel 20^Output'}
	bSound_2S1_HL1			AT%Q*	:BOOL;
//---------------------------------------------------------------------------------------------------------------//
// 4 цвета + сирена на стойке стеллажа h=3000мм Конвейер 3
{attribute 'TcLinkTo' := 'TIID^Device 1 (EtherCAT)^Term 1 (EK1200)^Term 11 (EK1122)^Term 12 (EK1100)^Term 24 (EK1322)^Box 1 (EPP2339-0021) X3^Channel 29^Output'}
	bRed_3S1HL1 			AT%Q*	:BOOL;
{attribute 'TcLinkTo' := 'TIID^Device 1 (EtherCAT)^Term 1 (EK1200)^Term 11 (EK1122)^Term 12 (EK1100)^Term 24 (EK1322)^Box 1 (EPP2339-0021) X3^Channel 30^Output'}
	bGreen_3S1HL1 			AT%Q*	:BOOL;
{attribute 'TcLinkTo' := 'TIID^Device 1 (EtherCAT)^Term 1 (EK1200)^Term 11 (EK1122)^Term 12 (EK1100)^Term 24 (EK1322)^Box 1 (EPP2339-0021) X3^Channel 31^Output'}
	bYellow_3S1HL1 	 		AT%Q*	:BOOL;
{attribute 'TcLinkTo' := 'TIID^Device 1 (EtherCAT)^Term 1 (EK1200)^Term 11 (EK1122)^Term 12 (EK1100)^Term 24 (EK1322)^Box 1 (EPP2339-0021) X3^Channel 32^Output'}
	bBlue_3S1HL1 			AT%Q*	:BOOL;
{attribute 'TcLinkTo' := 'TIID^Device 1 (EtherCAT)^Term 1 (EK1200)^Term 11 (EK1122)^Term 12 (EK1100)^Term 24 (EK1322)^Box 1 (EPP2339-0021) X3^Channel 28^Output'}
	bSound_3S1HL1			AT%Q*	:BOOL;
//---------------------------------------------------------------------------------------------------------------//
// 4 цвета + сирена на стойке стеллажа h=3000мм Конвейер 3
{attribute 'TcLinkTo' := 'TIID^Device 1 (EtherCAT)^Term 1 (EK1200)^Term 11 (EK1122)^Term 12 (EK1100)^Term 24 (EK1322)^Box 3 (EPP2339-0021) X3^Channel 21^Output'}
	bRed_3S1_HL1 			AT%Q*	:BOOL;
{attribute 'TcLinkTo' := 'TIID^Device 1 (EtherCAT)^Term 1 (EK1200)^Term 11 (EK1122)^Term 12 (EK1100)^Term 24 (EK1322)^Box 3 (EPP2339-0021) X3^Channel 22^Output'}
	bGreen_3S1_HL1 			AT%Q*	:BOOL;
{attribute 'TcLinkTo' := 'TIID^Device 1 (EtherCAT)^Term 1 (EK1200)^Term 11 (EK1122)^Term 12 (EK1100)^Term 24 (EK1322)^Box 3 (EPP2339-0021) X3^Channel 23^Output'}
	bYellow_3S1_HL1 	 	AT%Q*	:BOOL;
{attribute 'TcLinkTo' := 'TIID^Device 1 (EtherCAT)^Term 1 (EK1200)^Term 11 (EK1122)^Term 12 (EK1100)^Term 24 (EK1322)^Box 3 (EPP2339-0021) X3^Channel 24^Output'}
	bBlue_3S1_HL1 			AT%Q*	:BOOL;
{attribute 'TcLinkTo' := 'TIID^Device 1 (EtherCAT)^Term 1 (EK1200)^Term 11 (EK1122)^Term 12 (EK1100)^Term 24 (EK1322)^Box 3 (EPP2339-0021) X3^Channel 20^Output'}
	bSound_3S1_HL1			AT%Q*	:BOOL;
//---------------------------------------------------------------------------------------------------------------//
// 4 цвета + сирена на стойке стеллажа h=3000мм Конвейер 4
{attribute 'TcLinkTo' := 'TIID^Device 1 (EtherCAT)^Term 1 (EK1200)^Term 11 (EK1122)^Term 12 (EK1100)^Term 24 (EK1322)^Box 4 (EPP2339-0021) X4^Channel 24^Output'}
	bRed_4S1HL1 			AT%Q*	:BOOL;
{attribute 'TcLinkTo' := 'TIID^Device 1 (EtherCAT)^Term 1 (EK1200)^Term 11 (EK1122)^Term 12 (EK1100)^Term 24 (EK1322)^Box 4 (EPP2339-0021) X4^Channel 30^Output'}
	bGreen_4S1HL1 			AT%Q*	:BOOL;
{attribute 'TcLinkTo' := 'TIID^Device 1 (EtherCAT)^Term 1 (EK1200)^Term 11 (EK1122)^Term 12 (EK1100)^Term 24 (EK1322)^Box 4 (EPP2339-0021) X4^Channel 31^Output'}
	bYellow_4S1HL1 	 		AT%Q*	:BOOL;
{attribute 'TcLinkTo' := 'TIID^Device 1 (EtherCAT)^Term 1 (EK1200)^Term 11 (EK1122)^Term 12 (EK1100)^Term 24 (EK1322)^Box 4 (EPP2339-0021) X4^Channel 32^Output'}
	bBlue_4S1HL1 			AT%Q*	:BOOL;
{attribute 'TcLinkTo' := 'TIID^Device 1 (EtherCAT)^Term 1 (EK1200)^Term 11 (EK1122)^Term 12 (EK1100)^Term 24 (EK1322)^Box 4 (EPP2339-0021) X4^Channel 28^Output'}
	bSound_4S1HL1			AT%Q*	:BOOL;
//---------------------------------------------------------------------------------------------------------------//
// 4 цвета + сирена на стойке стеллажа h=3000мм Конвейер 4
{attribute 'TcLinkTo' := 'TIID^Device 1 (EtherCAT)^Term 1 (EK1200)^Term 11 (EK1122)^Term 12 (EK1100)^Term 24 (EK1322)^Box 6 (EPP2339-0021) X4^Channel 21^Output'}
	bRed_4S1_HL1 			AT%Q*	:BOOL;
{attribute 'TcLinkTo' := 'TIID^Device 1 (EtherCAT)^Term 1 (EK1200)^Term 11 (EK1122)^Term 12 (EK1100)^Term 24 (EK1322)^Box 6 (EPP2339-0021) X4^Channel 22^Output'}
	bGreen_4S1_HL1 			AT%Q*	:BOOL;
{attribute 'TcLinkTo' := 'TIID^Device 1 (EtherCAT)^Term 1 (EK1200)^Term 11 (EK1122)^Term 12 (EK1100)^Term 24 (EK1322)^Box 6 (EPP2339-0021) X4^Channel 23^Output'}
	bYellow_4S1_HL1 	 	AT%Q*	:BOOL;
{attribute 'TcLinkTo' := 'TIID^Device 1 (EtherCAT)^Term 1 (EK1200)^Term 11 (EK1122)^Term 12 (EK1100)^Term 24 (EK1322)^Box 6 (EPP2339-0021) X4^Channel 24^Output'}
	bBlue_4S1_HL1 			AT%Q*	:BOOL;
{attribute 'TcLinkTo' := 'TIID^Device 1 (EtherCAT)^Term 1 (EK1200)^Term 11 (EK1122)^Term 12 (EK1100)^Term 24 (EK1322)^Box 6 (EPP2339-0021) X4^Channel 20^Output'}
	bSound_4S1_HL1			AT%Q*	:BOOL;

	bNotReadyCC1_HLA1_Red  			:BOOL;		// Красный цвет
	bNotReadyCC1_HLA1_Yellow        :BOOL;		// Желтый цвет
	bNotReadyCC1_HLA1_Green         :BOOL;		// Зелёный цвет
	bNotReadyCC1_HLA1_Blue          :BOOL;		// Синий цвет
	bNotReadyCC1_HLA1_Sound         :BOOL;		// Звуковой сигнал
END_VAR

// ---- GVLs/GVL_LoadData_1.TcGVL
VAR_GLOBAL
	
	sScanID_1			: STRING;
	bRequestID_1		: BOOL;
	bReadScan_1			: BOOL;
	sWeight_1			: STRING;
	bRequestWeight_1	: BOOL;
	bReadWeight_1		: BOOL;
	
	sScanID_2			: STRING;
	bRequestID_2		: BOOL;
	bReadScan_2			: BOOL;
	sWeight_2			: STRING;
	bRequestWeight_2	: BOOL;
	bReadWeight_2		: BOOL;
	
	sScanID_3			: STRING;
	bRequestID_3		: BOOL;
	bReadScan_3			: BOOL;
	sWeight_3			: STRING;
	bRequestWeight_3	: BOOL;
	bReadWeight_3		: BOOL;
	
	sScanID_4			: STRING;
	bRequestID_4		: BOOL;
	bReadScan_4			: BOOL;
	sWeight_4			: STRING;
	bRequestWeight_4	: BOOL;
	bReadWeight_4		: BOOL;
	
	bOverflow_CTU_ID1		:BOOL;		//Переполнение счетчика несчитываний ID 1
	bOverflow_CTU_Weight1	:BOOL;		//Переполнение счетчика несчитываний весов 1
	
	bOverflow_CTU_ID2		:BOOL;		//Переполнение счетчика несчитываний ID 2
	bOverflow_CTU_Weight2	:BOOL;		//Переполнение счетчика несчитываний весов 2
	
	bOverflow_CTU_ID3		:BOOL;		//Переполнение счетчика несчитываний ID 3
	bOverflow_CTU_Weight3	:BOOL;		//Переполнение счетчика несчитываний весов 3
	
	bOverflow_CTU_ID4		:BOOL;		//Переполнение счетчика несчитываний ID 4
	bOverflow_CTU_Weight4	:BOOL;		//Переполнение счетчика несчитываний весов 4
	
	sMessageOut1:T_MaxString;
	bMessageReady1:BOOL;
	
	sMessageOut2:T_MaxString;
	bMessageReady2:BOOL;
	sMessageOut3:T_MaxString;
	bMessageReady3:BOOL;
	sMessageOut4:T_MaxString;
	bMessageReady4:BOOL;
	
END_VAR
VAR_GLOBAL  PERSISTENT
		stLoadS4_1		: ST_LoadData;
		stLoadS4_5_1	: ST_LoadData;
		stLoadS5_1		: ST_LoadData;
		stLoadS5_6_1	: ST_LoadData;
		stLoadS6_1		: ST_LoadData;
		
		stLoadS4_2		: ST_LoadData;
		stLoadS4_5_2	: ST_LoadData;
		stLoadS5_2		: ST_LoadData;
		stLoadS5_6_2	: ST_LoadData;
		stLoadS6_2		: ST_LoadData;
		
		stLoadS4_3		: ST_LoadData;
		stLoadS4_5_3	: ST_LoadData;
		stLoadS5_3		: ST_LoadData;
		stLoadS5_6_3	: ST_LoadData;
		stLoadS6_3		: ST_LoadData;
		
		
		stLoadS4_4		: ST_LoadData;
		stLoadS4_5_4	: ST_LoadData;
		stLoadS5_4		: ST_LoadData;
		stLoadS5_6_4	: ST_LoadData;
		stLoadS6_4		: ST_LoadData;
		
			
		
		
END_VAR

// ---- POUs/MAIN.TcPOU
PROGRAM MAIN
VAR
	fbPulse1 		:BLINK;
	fbPulse2 		:BLINK;
	fbPulse3 		:BLINK;
	fbPulse4 		:BLINK;
	fbPuls_Move  	:Puls;
	fbPuls_Reverse  :Puls;
	fbAlarmSound 	:PULS;
	fbButtAuto1 	:FB_ButtonToggle;
	fbButtManu1 	:FB_ButtonToggle;
	fbButtStop1 	:FB_ButtonToggle;
	fbButtReverse1 	:FB_ButtonToggle;
	fbStartAutomat1 :R_TRIG;
	fbStartSound1	:TP;	
	fbTimerStart1 	:TON;
	fbPuls 			:FB_Puls;
	
	fbButtAuto2 	:FB_ButtonToggle;
	fbButtManu2 	:FB_ButtonToggle;
	fbButtStop2 	:FB_ButtonToggle;
	fbButtReverse2 	:FB_ButtonToggle;
	fbStartAutomat2 :R_TRIG;
	fbStartSound2	:TP;	
	fbTimerStart2 	:TON;
	
	fbButtAuto3 	:FB_ButtonToggle;
	fbButtManu3 	:FB_ButtonToggle;
	fbButtStop3 	:FB_ButtonToggle;
	fbButtReverse3 	:FB_ButtonToggle;
	fbStartAutomat3 :R_TRIG;
	fbStartSound3	:TP;	
	fbTimerStart3 	:TON;
	
	fbButtAuto4 	:FB_ButtonToggle;
	fbButtManu4 	:FB_ButtonToggle;
	fbButtStop4 	:FB_ButtonToggle;
	fbButtReverse4 	:FB_ButtonToggle;
	fbStartAutomat4 :R_TRIG;
	fbStartSound4	:TP;	
	fbTimerStart4 	:TON;
	test:BOOL;
END_VAR


	TCP_IP();
	ACT_Drive();
	ACT_Light();
	Alarm_conv_1();
	Alarm_conv_2();
	Alarm_conv_3();
	Alarm_conv_4();
	Alarm_conv_General();
	ACT_Conversion();
	
	Exchange_WMS();
	

	fbPuls_Move(Period :=T#1S);
	fbPuls_Reverse(Period :=T#1.5S);
//----------------------------------------------------------------------------//
	//IF b_1K1_1 THEN bDirect1 := TRUE;
//		ELSE bDirect1 := FALSE;
//	END_IF
	
ConvLine1(bAutomat:=bAutomat1, bManual:=bManual1, bStop:=bStop1, bReset:= bReset1, bDirect:=bDirect1, bReverse:=bReverse1, bBuffering:=bBuffering1);

	fbButtAuto1(bButt := bButtAuto1 AND NOT bManual1 AND NOT bStop1, bReset := bReset1 OR bAlarm1);
	fbStartSound1 (IN :=fbButtAuto1.bOutB, PT :=T#3S);																
	bSound1 := fbStartSound1.Q;
	
    fbStartAutomat1(CLK := fbButtAuto1.bOutB AND NOT bSound1);

IF  fbStartAutomat1.Q THEN bStartAutomat1 := TRUE;
END_IF
		
	bAutomat1 := fbButtAuto1.bOutB  AND NOT bStartAutomat1 AND NOT bSound1 AND NOT bStop1;
	fbPuls(tPeriod := T#0.5S);

	fbButtManu1(bButt := bButtManu1 AND NOT  bAutomat1 AND NOT bSound1, bReset := bReset1 OR bAlarm1);
	bManual1 := fbButtManu1.bOutB;

//	fbButtReverse1(bButt := bButtReverse1 AND NOT b_1KM1_1, bReset := bReset1 OR bAlarm1);
//	bReverse1 := fbButtReverse1.bOutB;

	fbButtStop1(bButt := bButtStop1 OR bAlarm1, bReset := bReset1);
	bStop1 := fbButtStop1.bOutB ;
    	
	fbTimerStart1 (IN := bStartAutomat1, PT := T#1S);

IF NOT bStop1 AND fbTimerStart1.Q AND NOT 
  ( bDrive1s01M1 OR bDrive1s02M1 OR bDrive1s03M1 OR 
	bDrive1s04M1 OR bDrive1s05M1 OR bDrive1s06M1 OR 
	bDrive1s01M1Rev OR bDrive1s02M1Rev OR bDrive1s03M1Rev OR 
	bDrive1s04M1Rev OR bDrive1s05M1Rev OR bDrive1s06M1Rev )
THEN bStartAutomat1 := FALSE;
END_IF

IF bReset1 THEN bAutomat1 := FALSE; bManual1 := FALSE; bStop1 := FALSE; bStartAutomat1 := FALSE;
END_IF

fbpulse1(ENABLE := bStartAutomat1 OR bSound1,TIMELOW := T#500MS, TIMEHIGH:=T#500MS);
//Светофоры первого конвейера
bGreen_1S1HL1  := bAutomat1 AND NOT bManual1 AND NOT bAlarm1 AND NOT bSound1 AND b_1AS1 OR fbpulse1.OUT;
bGreen_1S1_HL1 := bAutomat1 AND NOT bManual1 AND NOT bAlarm1 AND NOT bSound1 AND b_1AS1 OR fbpulse1.OUT;

bYellow_1S1HL1 := NOT bAutomat1 AND bManual1 AND NOT bAlarm1;
bYellow_1S1_HL1:= NOT bAutomat1 AND bManual1 AND NOT bAlarm1;
//---------------------------------------------------------------------------------------------------//

	//IF b_2K1_1 THEN bDirect2 := TRUE;
//		ELSE bDirect2 := FALSE;
//	END_IF
	
ConvLine2(bAutomat:=bAutomat2, bManual:=bManual2, bStop:=bStop2, bReset:= bReset2, bDirect:=bDirect2, bReverse:=bReverse2, bBuffering:=bBuffering2);

	fbButtAuto2(bButt := bButtAuto2 AND NOT bManual2, bReset := bReset2 OR bAlarm2);
	fbStartSound2 (IN :=fbButtAuto2.bOutB, PT :=T#3S);																
	bSound2 := fbStartSound2.Q  ;
	
    fbStartAutomat2(CLK := fbButtAuto2.bOutB AND NOT bSound2);

IF  fbStartAutomat2.Q THEN bStartAutomat2 := TRUE;
END_IF
		
	bAutomat2 := fbButtAuto2.bOutB  AND NOT bStartAutomat2 AND NOT bSound2;
	fbPuls(tPeriod := T#0.5S);

	fbButtManu2(bButt := bButtManu2 AND NOT  bAutomat2, bReset := bReset2 OR bAlarm2);
	bManual2 := fbButtManu2.bOutB;

	fbButtReverse2(bButt := bButtReverse2 AND NOT b_2KM1_1, bReset := bReset2 OR bAlarm2);
	bReverse2 := fbButtReverse2.bOutB;

	fbButtStop2(bButt := bButtStop2 OR bAlarm2, bReset := bReset2);
	bStop2 := fbButtStop2.bOutB ;
    	
	fbTimerStart2 (IN := bStartAutomat2, PT := T#1S);

IF NOT bStop2 AND fbTimerStart2.Q AND NOT 
  ( bDrive2s01M1 OR bDrive2s02M1 OR bDrive2s03M1 OR 
	bDrive2s04M1 OR bDrive2s05M1 OR bDrive2s06M1 OR 
	bDrive2s01M1Rev OR bDrive2s02M1Rev OR bDrive2s03M1Rev OR 
	bDrive2s04M1Rev OR bDrive2s05M1Rev OR bDrive2s06M1Rev )
THEN bStartAutomat2 := FALSE;
END_IF

IF bReset2 THEN bAutomat2 := FALSE; bManual2 := FALSE; bStop2 := FALSE; bStartAutomat2 := FALSE;
END_IF

fbpulse2(ENABLE := bStartAutomat2 OR bSound2,TIMELOW := T#500MS, TIMEHIGH:=T#500MS);
//Светофоры первого конвейера
bGreen_2S1HL1  := bAutomat2 AND NOT bManual2 AND NOT bAlarm2 AND NOT bSound2 AND b_2AS1 OR fbpulse2.OUT;
bGreen_2S1_HL1 := bAutomat2 AND NOT bManual2 AND NOT bAlarm2 AND NOT bSound2 AND b_2AS1 OR fbpulse2.OUT;

bYellow_2S1HL1 := NOT bAutomat2 AND bManual2 AND NOT bAlarm2;
bYellow_2S1_HL1:= NOT bAutomat2 AND bManual2 AND NOT bAlarm2;
//---------------------------------------------------------------------------------------------------//

//	IF b_3K1_1 THEN bDirect3 := TRUE;
//		ELSE bDirect3 := FALSE;
//	END_IF
	
ConvLine3(bAutomat:=bAutomat3, bManual:=bManual3, bStop:=bStop3, bReset:= bReset3, bDirect:=bDirect3, bReverse:=bReverse3, bBuffering:=bBuffering3);

	fbButtAuto3(bButt := bButtAuto3 AND NOT bManual3, bReset := bReset3 OR bAlarm3);
	fbStartSound3 (IN :=fbButtAuto3.bOutB, PT :=T#3S);																
	bSound3 := fbStartSound3.Q  ;
	
    fbStartAutomat3(CLK := fbButtAuto3.bOutB AND NOT bSound3);

IF  fbStartAutomat3.Q THEN bStartAutomat3 := TRUE;
END_IF
		
	bAutomat3 := fbButtAuto3.bOutB  AND NOT bStartAutomat3 AND NOT bSound3;
	fbPuls(tPeriod := T#0.5S);

	fbButtManu3(bButt := bButtManu3 AND NOT  bAutomat3, bReset := bReset3 OR bAlarm3);
	bManual3 := fbButtManu3.bOutB;

	fbButtReverse3(bButt := bButtReverse3 AND NOT b_3KM1_1, bReset := bReset3 OR bAlarm3);
	bReverse3 := fbButtReverse3.bOutB;

	fbButtStop3(bButt := bButtStop3 OR bAlarm3, bReset := bReset3);
	bStop3 := fbButtStop3.bOutB ;
    	
	fbTimerStart3 (IN := bStartAutomat3, PT := T#1S);

IF NOT bStop3 AND fbTimerStart3.Q AND NOT 
  ( bDrive3s01M1 OR bDrive3s02M1 OR bDrive3s03M1 OR 
	bDrive3s04M1 OR bDrive3s05M1 OR bDrive3s06M1 OR 
	bDrive3s01M1Rev OR bDrive3s02M1Rev OR bDrive3s03M1Rev OR 
	bDrive3s04M1Rev OR bDrive3s05M1Rev OR bDrive3s06M1Rev )
THEN bStartAutomat3 := FALSE;
END_IF

IF bReset3 THEN bAutomat3 := FALSE; bManual3 := FALSE; bStop3 := FALSE; bStartAutomat3 := FALSE;
END_IF

fbpulse3(ENABLE := bStartAutomat3 OR bSound3,TIMELOW := T#500MS, TIMEHIGH:=T#500MS);
//Светофоры первого конвейера
bGreen_3S1HL1  := bAutomat3 AND NOT bManual3 AND NOT bAlarm3 AND NOT bSound3 OR fbpulse3.OUT;
bGreen_3S1_HL1 := bAutomat3 AND NOT bManual3 AND NOT bAlarm3 AND NOT bSound3 OR fbpulse3.OUT;

bYellow_3S1HL1 := NOT bAutomat3 AND bManual3 AND NOT bAlarm3;
bYellow_3S1_HL1:= NOT bAutomat3 AND bManual3 AND NOT bAlarm3;
//---------------------------------------------------------------------------------------------------//

//	IF b_4K1_1 THEN bDirect4 := TRUE;
//		ELSE bDirect4 := FALSE;
//	END_IF
	
ConvLine4(bAutomat:=bAutomat4, bManual:=bManual4, bStop:=bStop4, bReset:= bReset4, bDirect:=bDirect4, bReverse:=bReverse4, bBuffering:=bBuffering4);

	fbButtAuto4(bButt := bButtAuto4 AND NOT bManual4, bReset := bReset4 OR bAlarm4);
	fbStartSound4 (IN :=fbButtAuto4.bOutB, PT :=T#3S);																
	bSound4 := fbStartSound4.Q  ;
	
    fbStartAutomat4(CLK := fbButtAuto4.bOutB AND NOT bSound4);

IF  fbStartAutomat4.Q THEN bStartAutomat4 := TRUE;
END_IF
		
